QRS_NEXT_CUT()
PTP {E1 33657.188,E2 33657.188}
PTP {X 0,Y 759.907,A -85,B 0,C 180,E1 33657.188,E2 33657.188,E3 0,E4 0,E5 0,E6 0}
QRS_SPEED_INIT()
LIN {X 0,Y 759.907,Z 1240.5,A -85,B 0,C 180,E1 33657.188,E2 33657.188,E3 0,E4 0,E5 0,E6 0} C_VEL
LIN {X 0,Y 759.907,Z 488.645,A -85,B 0,C 180,E1 33657.188,E2 33657.188} C_VEL
LIN {X 0,Y 759.907,Z 480.571,A -85,B 0,C 180,E1 33657.188,E2 33657.188} C_VEL
LIN {X 0,Y 759.906,Z 478.571,A -85,B 0,C 180,E1 33657.037,E2 33657.037} C_VEL
LIN {X 0,Y 759.876,Z 478.573,A -85,B 0,C 180,E1 33654.26,E2 33654.26} C_VEL
LIN {X 0,Y 759.887,Z 478.566,A -85,B 0,C 180,E1 33651.525,E2 33651.525} C_VEL
LIN {X 0,Y 759.914,Z 478.576,A -85,B 0,C 180,E1 33648.54,E2 33648.54} C_VEL
LIN {X 0,Y 759.87,Z 478.57,A -85,B 0,C 180,E1 33645.755,E2 33645.755} C_VEL
LIN {X 0,Y 759.91,Z 478.564,A -85,B 0,C 180,E1 33643.016,E2 33643.016} C_VEL
LIN {X 0,Y 759.902,Z 478.576,A -85,B 0,C 180,E1 33640.075,E2 33640.075} C_VEL
LIN {X 0,Y 759.878,Z 478.567,A -85,B 0,C 180,E1 33637.277,E2 33637.277} C_VEL
LIN {X 0,Y 759.903,Z 478.568,A -85,B 0,C 180,E1 33634.504,E2 33634.504} C_VEL
LIN {X 0,Y 759.886,Z 478.574,A -85,B 0,C 180,E1 33631.639,E2 33631.639} C_VEL
LIN {X 0,Y 759.901,Z 478.565,A -85,B 0,C 180,E1 33628.773,E2 33628.773} C_VEL
LIN {X 0,Y 759.911,Z 478.578,A -85,B 0,C 180,E1 33625.72,E2 33625.72} C_VEL
LIN {X 0,Y 759.88,Z 478.567,A -85,B 0,C 180,E1 33622.881,E2 33622.881} C_VEL
LIN {X 0,Y 759.901,Z 478.568,A -85,B 0,C 180,E1 33620.094,E2 33620.094} C_VEL
LIN {X 0,Y 759.892,Z 478.574,A -85,B 0,C 180,E1 33617.237,E2 33617.237} C_VEL
LIN {X 0,Y 759.907,Z 478.564,A -85,B 0,C 180,E1 33614.32,E2 33614.32} C_VEL
LIN {X 0,Y 759.912,Z 478.577,A -85,B 0,C 180,E1 33611.238,E2 33611.238} C_VEL
LIN {X 0,Y 759.89,Z 478.567,A -85,B 0,C 180,E1 33608.349,E2 33608.349} C_VEL
LIN {X 0,Y 759.896,Z 478.575,A -85,B 0,C 180,E1 33605.561,E2 33605.561} C_VEL
LIN {X 0,Y 759.907,Z 478.918,A -85,B 0,C 180,E1 33605.243,E2 33605.243} C_VEL
LIN {X 0,Y 759.889,Z 515.935,A -85,B 0,C 180,E1 33603.007,E2 33603.007} C_VEL
LIN {X 0,Y 759.89,Z 560.734,A -85,B 0,C 180,E1 33600.393,E2 33600.393} C_VEL
LIN {X 0,Y 759.909,Z 611.611,A -85,B 0,C 180,E1 33597.505,E2 33597.505} C_VEL
LIN {X 0,Y 759.897,Z 651.654,A -85,B 0,C 180,E1 33595.304,E2 33595.304} C_VEL
LIN {X 0,Y 759.918,Z 925.114,A -85,B 0,C 180,E1 33592.529,E2 33592.529} C_VEL
LIN {X 0,Y 759.905,Z 958.983,A -85,B 0,C 180,E1 33592.158,E2 33592.158} C_VEL
LIN {X 0,Y 759.914,Z 979.59,A -85,B 0,C 180,E1 33591.8,E2 33591.8} C_VEL
LIN {X 0,Y 759.905,Z 1001.056,A -85,B 0,C 180,E1 33591.294,E2 33591.294} C_VEL
LIN {X 0,Y 759.917,Z 1021.303,A -85,B 0,C 180,E1 33590.686,E2 33590.686} C_VEL
LIN {X 0,Y 759.918,Z 1040.609,A -85,B 0,C 180,E1 33589.964,E2 33589.964} C_VEL
LIN {X 0,Y 759.917,Z 1060.421,A -85,B 0,C 180,E1 33589.084,E2 33589.084} C_VEL
LIN {X 0,Y 759.915,Z 1079.363,A -85,B 0,C 180,E1 33588.09,E2 33588.09} C_VEL
LIN {X 0,Y 759.915,Z 1097.201,A -85,B 0,C 180,E1 33586.983,E2 33586.983} C_VEL
LIN {X 0,Y 759.915,Z 1114.106,A -85,B 0,C 180,E1 33585.766,E2 33585.766} C_VEL
LIN {X 0,Y 759.917,Z 1129.971,A -85,B 0,C 180,E1 33584.436,E2 33584.436} C_VEL
LIN {X 0,Y 759.906,Z 1143.922,A -85,B 0,C 180,E1 33583.08,E2 33583.08} C_VEL
LIN {X 0,Y 759.906,Z 1156.086,A -85,B 0,C 180,E1 33581.691,E2 33581.691} C_VEL
LIN {X 0,Y 759.908,Z 1167.502,A -85,B 0,C 180,E1 33580.155,E2 33580.155} C_VEL
LIN {X 0,Y 759.913,Z 1177.015,A -85,B 0,C 180,E1 33578.627,E2 33578.627} C_VEL
LIN {X 0,Y 759.917,Z 1184.669,A -85,B 0,C 180,E1 33577.105,E2 33577.105} C_VEL
LIN {X 0,Y 759.909,Z 1191.249,A -85,B 0,C 180,E1 33575.436,E2 33575.436} C_VEL
LIN {X 0,Y 759.909,Z 1195.896,A -85,B 0,C 180,E1 33573.848,E2 33573.848} C_VEL
LIN {X 0,Y 759.914,Z 1198.939,A -85,B 0,C 180,E1 33572.187,E2 33572.187} C_VEL
LIN {X 0,Y 759.901,Z 1200.339,A -85,B 0,C 180,E1 33570.528,E2 33570.528} C_VEL
LIN {X 0,Y 759.911,Z 1200.186,A -85,B 0,C 180,E1 33568.945,E2 33568.945} C_VEL
LIN {X 0,Y 759.913,Z 1198.291,A -85,B 0,C 180,E1 33567.285,E2 33567.285} C_VEL
LIN {X 0,Y 759.916,Z 1194.725,A -85,B 0,C 180,E1 33565.623,E2 33565.623} C_VEL
LIN {X 0,Y 759.904,Z 1189.757,A -85,B 0,C 180,E1 33564.034,E2 33564.034} C_VEL
LIN {X 0,Y 759.899,Z 1182.966,A -85,B 0,C 180,E1 33562.439,E2 33562.439} C_VEL
LIN {X 0,Y 759.909,Z 1174.405,A -85,B 0,C 180,E1 33560.839,E2 33560.839} C_VEL
LIN {X 0,Y 759.908,Z 1164.458,A -85,B 0,C 180,E1 33559.308,E2 33559.308} C_VEL
LIN {X 0,Y 759.917,Z 1152.996,A -85,B 0,C 180,E1 33557.847,E2 33557.847} C_VEL
LIN {X 0,Y 759.915,Z 1140.229,A -85,B 0,C 180,E1 33556.455,E2 33556.455} C_VEL
LIN {X 0,Y 759.914,Z 1126.191,A -85,B 0,C 180,E1 33555.133,E2 33555.133} C_VEL
LIN {X 0,Y 759.911,Z 1110.315,A -85,B 0,C 180,E1 33553.85,E2 33553.85} C_VEL
LIN {X 0,Y 759.911,Z 1093.753,A -85,B 0,C 180,E1 33552.701,E2 33552.701} C_VEL
LIN {X 0,Y 759.917,Z 1075.204,A -85,B 0,C 180,E1 33551.592,E2 33551.592} C_VEL
LIN {X 0,Y 759.917,Z 1056.495,A -85,B 0,C 180,E1 33550.635,E2 33550.635} C_VEL
LIN {X 0,Y 759.92,Z 1036.873,A -85,B 0,C 180,E1 33549.795,E2 33549.795} C_VEL
LIN {X 0,Y 759.916,Z 1016.314,A -85,B 0,C 180,E1 33549.066,E2 33549.066} C_VEL
LIN {X 0,Y 759.911,Z 995.942,A -85,B 0,C 180,E1 33548.478,E2 33548.478} C_VEL
LIN {X 0,Y 759.909,Z 974.842,A -85,B 0,C 180,E1 33548.017,E2 33548.017} C_VEL
LIN {X 0,Y 759.907,Z 952.592,A -85,B 0,C 180,E1 33547.671,E2 33547.671} C_VEL
LIN {X 0,Y 759.898,Z 670.991,A -85,B 0,C 180,E1 33544.808,E2 33544.808} C_VEL
LIN {X 0,Y 759.898,Z 651.373,A -85,B 0,C 180,E1 33544.6,E2 33544.6} C_VEL
LIN {X 0,Y 759.905,Z 601.06,A -85,B 0,C 180,E1 33541.812,E2 33541.812} C_VEL
LIN {X 0,Y 759.918,Z 552.419,A -85,B 0,C 180,E1 33539.039,E2 33539.039} C_VEL
LIN {X 0,Y 759.919,Z 505.108,A -85,B 0,C 180,E1 33536.261,E2 33536.261} C_VEL
LIN {X 0,Y 759.908,Z 478.918,A -85,B 0,C 180,E1 33534.667,E2 33534.667} C_VEL
LIN {X 0,Y 759.908,Z 478.57,A -85,B 0,C 180,E1 33534.149,E2 33534.149} C_VEL
LIN {X 0,Y 759.874,Z 478.571,A -85,B 0,C 180,E1 33531.317,E2 33531.317} C_VEL
LIN {X 0,Y 759.914,Z 478.576,A -85,B 0,C 180,E1 33528.561,E2 33528.561} C_VEL
LIN {X 0,Y 759.894,Z 478.566,A -85,B 0,C 180,E1 33525.573,E2 33525.573} C_VEL
LIN {X 0,Y 759.884,Z 478.573,A -85,B 0,C 180,E1 33522.759,E2 33522.759} C_VEL
LIN {X 0,Y 759.904,Z 478.569,A -85,B 0,C 180,E1 33519.907,E2 33519.907} C_VEL
LIN {X 0,Y 759.877,Z 478.567,A -85,B 0,C 180,E1 33517.119,E2 33517.119} C_VEL
LIN {X 0,Y 759.895,Z 478.576,A -85,B 0,C 180,E1 33514.367,E2 33514.367} C_VEL
LIN {X 0,Y 759.91,Z 478.564,A -85,B 0,C 180,E1 33511.315,E2 33511.315} C_VEL
LIN {X 0,Y 759.868,Z 478.571,A -85,B 0,C 180,E1 33508.619,E2 33508.619} C_VEL
LIN {X 0,Y 759.912,Z 478.576,A -85,B 0,C 180,E1 33505.845,E2 33505.845} C_VEL
LIN {X 0,Y 759.891,Z 478.565,A -85,B 0,C 180,E1 33502.92,E2 33502.92} C_VEL
LIN {X 0,Y 759.874,Z 478.573,A -85,B 0,C 180,E1 33500.167,E2 33500.167} C_VEL
LIN {X 0,Y 759.906,Z 478.572,A -85,B 0,C 180,E1 33497.379,E2 33497.379} C_VEL
LIN {X 0,Y 759.878,Z 478.567,A -85,B 0,C 180,E1 33494.556,E2 33494.556} C_VEL
LIN {X 0,Y 759.877,Z 478.574,A -85,B 0,C 180,E1 33491.846,E2 33491.846} C_VEL
LIN {X 0,Y 759.907,Z 478.569,A -85,B 0,C 180,E1 33489.009,E2 33489.009} C_VEL
LIN {X 0,Y 759.868,Z 478.568,A -85,B 0,C 180,E1 33486.194,E2 33486.194} C_VEL
LIN {X 0,Y 759.887,Z 478.575,A -85,B 0,C 180,E1 33483.47,E2 33483.47} C_VEL
LIN {X 0,Y 759.91,Z 478.565,A -85,B 0,C 180,E1 33480.452,E2 33480.452} C_VEL
LIN {X 0,Y 759.861,Z 478.571,A -85,B 0,C 180,E1 33477.738,E2 33477.738} C_VEL
LIN {X 0,Y 759.909,Z 478.577,A -85,B 0,C 180,E1 33475.018,E2 33475.018} C_VEL
LIN {X 0,Y 759.888,Z 478.566,A -85,B 0,C 180,E1 33472.058,E2 33472.058} C_VEL
LIN {X 0,Y 759.861,Z 478.572,A -85,B 0,C 180,E1 33469.384,E2 33469.384} C_VEL
LIN {X 0,Y 759.918,Z 478.577,A -85,B 0,C 180,E1 33466.687,E2 33466.687} C_VEL
LIN {X 0,Y 759.876,Z 478.567,A -85,B 0,C 180,E1 33463.723,E2 33463.723} C_VEL
LIN {X 0,Y 759.86,Z 478.573,A -85,B 0,C 180,E1 33461.101,E2 33461.101} C_VEL
LIN {X 0,Y 759.915,Z 478.576,A -85,B 0,C 180,E1 33458.382,E2 33458.382} C_VEL
LIN {X 0,Y 759.877,Z 478.567,A -85,B 0,C 180,E1 33455.512,E2 33455.512} C_VEL
LIN {X 0,Y 759.856,Z 478.572,A -85,B 0,C 180,E1 33452.916,E2 33452.916} C_VEL
LIN {X 0,Y 759.904,Z 478.578,A -85,B 0,C 180,E1 33450.26,E2 33450.26} C_VEL
LIN {X 0,Y 759.883,Z 478.566,A -85,B 0,C 180,E1 33447.35,E2 33447.35} C_VEL
LIN {X 0,Y 759.853,Z 478.572,A -85,B 0,C 180,E1 33444.712,E2 33444.712} C_VEL
LIN {X 0,Y 759.914,Z 478.577,A -85,B 0,C 180,E1 33441.99,E2 33441.99} C_VEL
LIN {X 0,Y 759.874,Z 478.568,A -85,B 0,C 180,E1 33439.05,E2 33439.05} C_VEL
LIN {X 0,Y 759.851,Z 478.572,A -85,B 0,C 180,E1 33436.472,E2 33436.472} C_VEL
LIN {X 0,Y 759.912,Z 478.577,A -85,B 0,C 180,E1 33433.749,E2 33433.749} C_VEL
LIN {X 0,Y 759.875,Z 478.569,A -85,B 0,C 180,E1 33430.832,E2 33430.832} C_VEL
LIN {X 0,Y 759.849,Z 478.573,A -85,B 0,C 180,E1 33428.224,E2 33428.224} C_VEL
LIN {X 0,Y 759.889,Z 478.702,A -85,B 0,C 180,E1 33425.639,E2 33425.639} C_VEL
LIN {X 0,Y 759.917,Z 480.91,A -85,B 0,C 180,E1 33425.464,E2 33425.464} C_VEL
LIN {X 0,Y 759.915,Z 527.036,A -85,B 0,C 180,E1 33422.87,E2 33422.87} C_VEL
LIN {X 0,Y 759.912,Z 529.446,A -85,B 0,C 180,E1 33422.801,E2 33422.801} C_VEL
LIN {X 0,Y 759.891,Z 789.76,A -85,B 0,C 180,E1 33419.978,E2 33419.978} C_VEL
LIN {X 0,Y 759.917,Z 918.081,A -85,B 0,C 180,E1 33418.594,E2 33418.594} C_VEL
LIN {X 0,Y 759.894,Z 942.353,A -85,B 0,C 180,E1 33418.209,E2 33418.209} C_VEL
LIN {X 0,Y 759.901,Z 963.718,A -85,B 0,C 180,E1 33417.741,E2 33417.741} C_VEL
LIN {X 0,Y 759.907,Z 983.081,A -85,B 0,C 180,E1 33417.221,E2 33417.221} C_VEL
LIN {X 0,Y 759.919,Z 1005.766,A -85,B 0,C 180,E1 33416.49,E2 33416.49} C_VEL
LIN {X 0,Y 759.916,Z 1027.274,A -85,B 0,C 180,E1 33415.65,E2 33415.65} C_VEL
LIN {X 0,Y 759.918,Z 1046.636,A -85,B 0,C 180,E1 33414.784,E2 33414.784} C_VEL
LIN {X 0,Y 759.909,Z 1068.349,A -85,B 0,C 180,E1 33413.66,E2 33413.66} C_VEL
LIN {X 0,Y 759.913,Z 1086.397,A -85,B 0,C 180,E1 33412.594,E2 33412.594} C_VEL
LIN {X 0,Y 759.907,Z 1107.535,A -85,B 0,C 180,E1 33411.172,E2 33411.172} C_VEL
LIN {X 0,Y 759.916,Z 1124.895,A -85,B 0,C 180,E1 33409.844,E2 33409.844} C_VEL
LIN {X 0,Y 759.916,Z 1141.398,A -85,B 0,C 180,E1 33408.408,E2 33408.408} C_VEL
LIN {X 0,Y 759.898,Z 1155.953,A -85,B 0,C 180,E1 33406.984,E2 33406.984} C_VEL
LIN {X 0,Y 759.899,Z 1170.876,A -85,B 0,C 180,E1 33405.312,E2 33405.312} C_VEL
LIN {X 0,Y 759.9,Z 1182.583,A -85,B 0,C 180,E1 33403.813,E2 33403.813} C_VEL
LIN {X 0,Y 759.894,Z 1194.788,A -85,B 0,C 180,E1 33401.999,E2 33401.999} C_VEL
LIN {X 0,Y 759.907,Z 1203.557,A -85,B 0,C 180,E1 33400.462,E2 33400.462} C_VEL
LIN {X 0,Y 759.894,Z 1212.075,A -85,B 0,C 180,E1 33398.703,E2 33398.703} C_VEL
LIN {X 0,Y 759.918,Z 1218.727,A -85,B 0,C 180,E1 33396.953,E2 33396.953} C_VEL
LIN {X 0,Y 759.883,Z 1223.511,A -85,B 0,C 180,E1 33395.36,E2 33395.36} C_VEL
LIN {X 0,Y 759.919,Z 1227.559,A -85,B 0,C 180,E1 33393.47,E2 33393.47} C_VEL
LIN {X 0,Y 759.9,Z 1229.63,A -85,B 0,C 180,E1 33391.81,E2 33391.81} C_VEL
LIN {X 0,Y 759.92,Z 1230.5,A -85,B 0,C 180,E1 33390,E2 33390} C_VEL
LIN {X 0,Y 759.9,Z 1229.63,A -85,B 0,C 180,E1 33388.19,E2 33388.19} C_VEL
LIN {X 0,Y 759.919,Z 1227.559,A -85,B 0,C 180,E1 33386.53,E2 33386.53} C_VEL
LIN {X 0,Y 759.883,Z 1223.511,A -85,B 0,C 180,E1 33384.639,E2 33384.639} C_VEL
LIN {X 0,Y 759.918,Z 1218.726,A -85,B 0,C 180,E1 33383.047,E2 33383.047} C_VEL
LIN {X 0,Y 759.893,Z 1211.731,A -85,B 0,C 180,E1 33381.221,E2 33381.221} C_VEL
LIN {X 0,Y 759.907,Z 1203.557,A -85,B 0,C 180,E1 33379.538,E2 33379.538} C_VEL
LIN {X 0,Y 759.894,Z 1194.788,A -85,B 0,C 180,E1 33378.001,E2 33378.001} C_VEL
LIN {X 0,Y 759.9,Z 1182.583,A -85,B 0,C 180,E1 33376.187,E2 33376.187} C_VEL
LIN {X 0,Y 759.899,Z 1170.876,A -85,B 0,C 180,E1 33374.688,E2 33374.688} C_VEL
LIN {X 0,Y 759.898,Z 1155.953,A -85,B 0,C 180,E1 33373.016,E2 33373.016} C_VEL
LIN {X 0,Y 759.916,Z 1141.398,A -85,B 0,C 180,E1 33371.592,E2 33371.592} C_VEL
LIN {X 0,Y 759.911,Z 1123.375,A -85,B 0,C 180,E1 33370.036,E2 33370.036} C_VEL
LIN {X 0,Y 759.908,Z 1106.43,A -85,B 0,C 180,E1 33368.747,E2 33368.747} C_VEL
LIN {X 0,Y 759.914,Z 1086.396,A -85,B 0,C 180,E1 33367.406,E2 33367.406} C_VEL
LIN {X 0,Y 759.909,Z 1067.993,A -85,B 0,C 180,E1 33366.32,E2 33366.32} C_VEL
LIN {X 0,Y 759.919,Z 1045.919,A -85,B 0,C 180,E1 33365.183,E2 33365.183} C_VEL
LIN {X 0,Y 759.916,Z 1026.866,A -85,B 0,C 180,E1 33364.332,E2 33364.332} C_VEL
LIN {X 0,Y 759.918,Z 1004.811,A -85,B 0,C 180,E1 33363.475,E2 33363.475} C_VEL
LIN {X 0,Y 759.907,Z 982.044,A -85,B 0,C 180,E1 33362.749,E2 33362.749} C_VEL
LIN {X 0,Y 759.898,Z 962.099,A -85,B 0,C 180,E1 33362.219,E2 33362.219} C_VEL
LIN {X 0,Y 759.898,Z 937.439,A -85,B 0,C 180,E1 33361.702,E2 33361.702} C_VEL
LIN {X 0,Y 759.916,Z 916.368,A -85,B 0,C 180,E1 33361.384,E2 33361.384} C_VEL
LIN {X 0,Y 759.867,Z 652.343,A -85,B 0,C 180,E1 33358.541,E2 33358.541} C_VEL
LIN {X 0,Y 759.912,Z 527.915,A -85,B 0,C 180,E1 33357.174,E2 33357.174} C_VEL
LIN {X 0,Y 759.916,Z 481.69,A -85,B 0,C 180,E1 33354.58,E2 33354.58} C_VEL
LIN {X 0,Y 759.891,Z 478.77,A -85,B 0,C 180,E1 33354.377,E2 33354.377} C_VEL
LIN {X 0,Y 759.852,Z 478.574,A -85,B 0,C 180,E1 33351.893,E2 33351.893} C_VEL
LIN {X 0,Y 759.858,Z 478.57,A -85,B 0,C 180,E1 33349.357,E2 33349.357} C_VEL
LIN {X 0,Y 759.913,Z 478.57,A -85,B 0,C 180,E1 33346.579,E2 33346.579} C_VEL
LIN {X 0,Y 759.861,Z 478.573,A -85,B 0,C 180,E1 33343.747,E2 33343.747} C_VEL
LIN {X 0,Y 759.859,Z 478.57,A -85,B 0,C 180,E1 33341.144,E2 33341.144} C_VEL
LIN {X 0,Y 759.911,Z 478.569,A -85,B 0,C 180,E1 33338.354,E2 33338.354} C_VEL
LIN {X 0,Y 759.868,Z 478.574,A -85,B 0,C 180,E1 33335.564,E2 33335.564} C_VEL
LIN {X 0,Y 759.861,Z 478.568,A -85,B 0,C 180,E1 33332.92,E2 33332.92} C_VEL
LIN {X 0,Y 759.912,Z 478.569,A -85,B 0,C 180,E1 33330.175,E2 33330.175} C_VEL
LIN {X 0,Y 759.873,Z 478.574,A -85,B 0,C 180,E1 33327.338,E2 33327.338} C_VEL
LIN {X 0,Y 759.861,Z 478.569,A -85,B 0,C 180,E1 33324.737,E2 33324.737} C_VEL
LIN {X 0,Y 759.915,Z 478.567,A -85,B 0,C 180,E1 33322.024,E2 33322.024} C_VEL
LIN {X 0,Y 759.878,Z 478.575,A -85,B 0,C 180,E1 33319.126,E2 33319.126} C_VEL
LIN {X 0,Y 759.866,Z 478.569,A -85,B 0,C 180,E1 33316.434,E2 33316.434} C_VEL
LIN {X 0,Y 759.91,Z 478.568,A -85,B 0,C 180,E1 33313.7,E2 33313.7} C_VEL
LIN {X 0,Y 759.878,Z 478.574,A -85,B 0,C 180,E1 33310.846,E2 33310.846} C_VEL
LIN {X 0,Y 759.87,Z 478.568,A -85,B 0,C 180,E1 33308.17,E2 33308.17} C_VEL
LIN {X 0,Y 759.907,Z 478.57,A -85,B 0,C 180,E1 33305.361,E2 33305.361} C_VEL
LIN {X 0,Y 759.877,Z 478.574,A -85,B 0,C 180,E1 33302.564,E2 33302.564} C_VEL
LIN {X 0,Y 759.877,Z 478.567,A -85,B 0,C 180,E1 33299.849,E2 33299.849} C_VEL
LIN {X 0,Y 759.906,Z 478.571,A -85,B 0,C 180,E1 33297.037,E2 33297.037} C_VEL
LIN {X 0,Y 758.93,Z 478.703,A -85,B 0,C 180,E1 33296.456,E2 33296.456} C_VEL
LIN {X 0,Y 752.51,Z 479.501,A -85,B 0,C 180,E1 33294.83,E2 33294.83} C_VEL
LIN {X 0,Y 751.949,Z 479.563,A -85,B 0,C 180,E1 33294.407,E2 33294.407} C_VEL
LIN {X 0,Y 751.942,Z 479.556,A -85,B 0,C 180,E1 33291.589,E2 33291.589} C_VEL
LIN {X 0,Y 751.967,Z 479.56,A -85,B 0,C 180,E1 33288.728,E2 33288.728} C_VEL
LIN {X 0,Y 751.934,Z 479.56,A -85,B 0,C 180,E1 33285.916,E2 33285.916} C_VEL
LIN {X 0,Y 751.972,Z 479.553,A -85,B 0,C 180,E1 33283.07,E2 33283.07} C_VEL
LIN {X 0,Y 751.957,Z 479.564,A -85,B 0,C 180,E1 33280.017,E2 33280.017} C_VEL
LIN {X 0,Y 751.942,Z 479.555,A -85,B 0,C 180,E1 33277.235,E2 33277.235} C_VEL
LIN {X 0,Y 751.964,Z 479.559,A -85,B 0,C 180,E1 33274.396,E2 33274.396} C_VEL
LIN {X 0,Y 751.943,Z 479.562,A -85,B 0,C 180,E1 33271.572,E2 33271.572} C_VEL
LIN {X 0,Y 751.964,Z 479.553,A -85,B 0,C 180,E1 33268.756,E2 33268.756} C_VEL
LIN {X 0,Y 751.968,Z 479.566,A -85,B 0,C 180,E1 33265.661,E2 33265.661} C_VEL
LIN {X 0,Y 751.948,Z 479.553,A -85,B 0,C 180,E1 33262.769,E2 33262.769} C_VEL
LIN {X 0,Y 751.961,Z 479.559,A -85,B 0,C 180,E1 33259.94,E2 33259.94} C_VEL
LIN {X 0,Y 751.95,Z 479.561,A -85,B 0,C 180,E1 33257.196,E2 33257.196} C_VEL
LIN {X 0,Y 751.974,Z 479.553,A -85,B 0,C 180,E1 33254.272,E2 33254.272} C_VEL
LIN {X 0,Y 751.967,Z 479.565,A -85,B 0,C 180,E1 33251.183,E2 33251.183} C_VEL
LIN {X 0,Y 751.964,Z 479.556,A -85,B 0,C 180,E1 33248.191,E2 33248.191} C_VEL
LIN {X 0,Y 751.982,Z 479.737,A -85,B 0,C 180,E1 33245.641,E2 33245.641} C_VEL
LIN {X 0,Y 752.908,Z 483.22,A -85,B 0,C 180,E1 33245.339,E2 33245.339} C_VEL
LIN {X 0,Y 752.739,Z 526.575,A -85,B 0,C 180,E1 33242.725,E2 33242.725} C_VEL
LIN {X 0,Y 752.644,Z 573.653,A -85,B 0,C 180,E1 33239.967,E2 33239.967} C_VEL
LIN {X 0,Y 752.503,Z 622.252,A -85,B 0,C 180,E1 33237.199,E2 33237.199} C_VEL
LIN {X 0,Y 752.525,Z 651.817,A -85,B 0,C 180,E1 33235.568,E2 33235.568} C_VEL
LIN {X 0,Y 752.566,Z 857.23,A -85,B 0,C 180,E1 33233.452,E2 33233.452} C_VEL
LIN {X 0,Y 752.494,Z 956.636,A -85,B 0,C 180,E1 33232.422,E2 33232.422} C_VEL
LIN {X 0,Y 752.461,Z 977.93,A -85,B 0,C 180,E1 33232.061,E2 33232.061} C_VEL
LIN {X 0,Y 752.403,Z 999.609,A -85,B 0,C 180,E1 33231.558,E2 33231.558} C_VEL
LIN {X 0,Y 752.372,Z 1019.992,A -85,B 0,C 180,E1 33230.946,E2 33230.946} C_VEL
LIN {X 0,Y 752.309,Z 1039.631,A -85,B 0,C 180,E1 33230.216,E2 33230.216} C_VEL
LIN {X 0,Y 752.24,Z 1059.632,A -85,B 0,C 180,E1 33229.327,E2 33229.327} C_VEL
LIN {X 0,Y 752.187,Z 1078.654,A -85,B 0,C 180,E1 33228.323,E2 33228.323} C_VEL
LIN {X 0,Y 752.125,Z 1096.369,A -85,B 0,C 180,E1 33227.22,E2 33227.22} C_VEL
LIN {X 0,Y 752.074,Z 1113.607,A -85,B 0,C 180,E1 33225.974,E2 33225.974} C_VEL
LIN {X 0,Y 752.028,Z 1128.683,A -85,B 0,C 180,E1 33224.711,E2 33224.711} C_VEL
LIN {X 0,Y 751.996,Z 1142.434,A -85,B 0,C 180,E1 33223.377,E2 33223.377} C_VEL
LIN {X 0,Y 751.967,Z 1154.812,A -85,B 0,C 180,E1 33221.972,E2 33221.972} C_VEL
LIN {X 0,Y 751.944,Z 1166.471,A -85,B 0,C 180,E1 33220.419,E2 33220.419} C_VEL
LIN {X 0,Y 751.93,Z 1176.168,A -85,B 0,C 180,E1 33218.873,E2 33218.873} C_VEL
LIN {X 0,Y 751.914,Z 1183.964,A -85,B 0,C 180,E1 33217.334,E2 33217.334} C_VEL
LIN {X 0,Y 751.9,Z 1190.492,A -85,B 0,C 180,E1 33215.724,E2 33215.724} C_VEL
LIN {X 0,Y 751.918,Z 1195.302,A -85,B 0,C 180,E1 33214.118,E2 33214.118} C_VEL
LIN {X 0,Y 751.911,Z 1198.606,A -85,B 0,C 180,E1 33212.439,E2 33212.439} C_VEL
LIN {X 0,Y 751.913,Z 1200.272,A -85,B 0,C 180,E1 33210.762,E2 33210.762} C_VEL
LIN {X 0,Y 751.913,Z 1200.254,A -85,B 0,C 180,E1 33209.086,E2 33209.086} C_VEL
LIN {X 0,Y 751.909,Z 1198.626,A -85,B 0,C 180,E1 33207.485,E2 33207.485} C_VEL
LIN {X 0,Y 751.918,Z 1195.338,A -85,B 0,C 180,E1 33205.806,E2 33205.806} C_VEL
LIN {X 0,Y 751.904,Z 1190.536,A -85,B 0,C 180,E1 33204.2,E2 33204.2} C_VEL
LIN {X 0,Y 751.911,Z 1184.025,A -85,B 0,C 180,E1 33202.589,E2 33202.589} C_VEL
LIN {X 0,Y 751.931,Z 1176.245,A -85,B 0,C 180,E1 33201.05,E2 33201.05} C_VEL
LIN {X 0,Y 751.945,Z 1166.555,A -85,B 0,C 180,E1 33199.504,E2 33199.504} C_VEL
LIN {X 0,Y 751.964,Z 1154.912,A -85,B 0,C 180,E1 33197.951,E2 33197.951} C_VEL
LIN {X 0,Y 751.997,Z 1142.549,A -85,B 0,C 180,E1 33196.545,E2 33196.545} C_VEL
LIN {X 0,Y 752.028,Z 1128.199,A -85,B 0,C 180,E1 33195.154,E2 33195.154} C_VEL
LIN {X 0,Y 752.071,Z 1112.734,A -85,B 0,C 180,E1 33193.868,E2 33193.868} C_VEL
LIN {X 0,Y 752.124,Z 1095.859,A -85,B 0,C 180,E1 33192.656,E2 33192.656} C_VEL
LIN {X 0,Y 752.189,Z 1078.106,A -85,B 0,C 180,E1 33191.557,E2 33191.557} C_VEL
LIN {X 0,Y 752.24,Z 1059.818,A -85,B 0,C 180,E1 33190.592,E2 33190.592} C_VEL
LIN {X 0,Y 752.309,Z 1039.849,A -85,B 0,C 180,E1 33189.703,E2 33189.703} C_VEL
LIN {X 0,Y 752.37,Z 1020.259,A -85,B 0,C 180,E1 33188.973,E2 33188.973} C_VEL
LIN {X 0,Y 752.403,Z 999.9,A -85,B 0,C 180,E1 33188.361,E2 33188.361} C_VEL
LIN {X 0,Y 752.461,Z 977.95,A -85,B 0,C 180,E1 33187.85,E2 33187.85} C_VEL
LIN {X 0,Y 752.494,Z 956.737,A -85,B 0,C 180,E1 33187.489,E2 33187.489} C_VEL
LIN {X 0,Y 752.563,Z 860.44,A -85,B 0,C 180,E1 33186.491,E2 33186.491} C_VEL
LIN {X 0,Y 752.538,Z 651.902,A -85,B 0,C 180,E1 33184.344,E2 33184.344} C_VEL
LIN {X 0,Y 752.461,Z 636.009,A -85,B 0,C 180,E1 33183.483,E2 33183.483} C_VEL
LIN {X 0,Y 752.565,Z 589.65,A -85,B 0,C 180,E1 33180.861,E2 33180.861} C_VEL
LIN {X 0,Y 752.723,Z 541.008,A -85,B 0,C 180,E1 33178.039,E2 33178.039} C_VEL
LIN {X 0,Y 752.872,Z 494.644,A -85,B 0,C 180,E1 33175.268,E2 33175.268} C_VEL
LIN {X 0,Y 752.808,Z 482.281,A -85,B 0,C 180,E1 33174.508,E2 33174.508} C_VEL
LIN {X 0,Y 751.986,Z 479.719,A -85,B 0,C 180,E1 33174.265,E2 33174.265} C_VEL
LIN {X 0,Y 751.937,Z 479.56,A -85,B 0,C 180,E1 33171.435,E2 33171.435} C_VEL
LIN {X 0,Y 751.973,Z 479.567,A -85,B 0,C 180,E1 33168.637,E2 33168.637} C_VEL
LIN {X 0,Y 751.96,Z 479.554,A -85,B 0,C 180,E1 33165.621,E2 33165.621} C_VEL
LIN {X 0,Y 751.944,Z 479.561,A -85,B 0,C 180,E1 33162.778,E2 33162.778} C_VEL
LIN {X 0,Y 751.965,Z 479.559,A -85,B 0,C 180,E1 33159.96,E2 33159.96} C_VEL
LIN {X 0,Y 751.939,Z 479.554,A -85,B 0,C 180,E1 33157.136,E2 33157.136} C_VEL
LIN {X 0,Y 751.961,Z 479.565,A -85,B 0,C 180,E1 33154.319,E2 33154.319} C_VEL
LIN {X 0,Y 751.963,Z 479.554,A -85,B 0,C 180,E1 33151.238,E2 33151.238} C_VEL
LIN {X 0,Y 751.934,Z 479.562,A -85,B 0,C 180,E1 33148.428,E2 33148.428} C_VEL
LIN {X 0,Y 751.966,Z 479.56,A -85,B 0,C 180,E1 33145.604,E2 33145.604} C_VEL
LIN {X 0,Y 751.939,Z 479.556,A -85,B 0,C 180,E1 33142.765,E2 33142.765} C_VEL
LIN {X 0,Y 751.949,Z 479.564,A -85,B 0,C 180,E1 33139.983,E2 33139.983} C_VEL
LIN {X 0,Y 751.973,Z 479.554,A -85,B 0,C 180,E1 33137.01,E2 33137.01} C_VEL
LIN {X 0,Y 751.927,Z 479.559,A -85,B 0,C 180,E1 33134.218,E2 33134.218} C_VEL
LIN {X 0,Y 751.977,Z 479.564,A -85,B 0,C 180,E1 33131.427,E2 33131.427} C_VEL
LIN {X 0,Y 751.948,Z 479.556,A -85,B 0,C 180,E1 33128.488,E2 33128.488} C_VEL
LIN {X 0,Y 751.929,Z 479.561,A -85,B 0,C 180,E1 33125.8,E2 33125.8} C_VEL
LIN {X 0,Y 751.972,Z 479.562,A -85,B 0,C 180,E1 33123.049,E2 33123.049} C_VEL
LIN {X 0,Y 751.937,Z 479.556,A -85,B 0,C 180,E1 33120.152,E2 33120.152} C_VEL
LIN {X 0,Y 751.93,Z 479.562,A -85,B 0,C 180,E1 33117.485,E2 33117.485} C_VEL
LIN {X 0,Y 751.97,Z 479.56,A -85,B 0,C 180,E1 33114.659,E2 33114.659} C_VEL
LIN {X 0,Y 751.934,Z 479.556,A -85,B 0,C 180,E1 33111.897,E2 33111.897} C_VEL
LIN {X 0,Y 751.932,Z 479.563,A -85,B 0,C 180,E1 33109.193,E2 33109.193} C_VEL
LIN {X 0,Y 751.972,Z 479.558,A -85,B 0,C 180,E1 33106.309,E2 33106.309} C_VEL
LIN {X 0,Y 751.924,Z 479.558,A -85,B 0,C 180,E1 33103.546,E2 33103.546} C_VEL
LIN {X 0,Y 751.933,Z 479.563,A -85,B 0,C 180,E1 33100.906,E2 33100.906} C_VEL
LIN {X 0,Y 751.978,Z 479.555,A -85,B 0,C 180,E1 33097.934,E2 33097.934} C_VEL
LIN {X 0,Y 751.919,Z 479.558,A -85,B 0,C 180,E1 33095.236,E2 33095.236} C_VEL
LIN {X 0,Y 751.936,Z 479.564,A -85,B 0,C 180,E1 33092.607,E2 33092.607} C_VEL
LIN {X 0,Y 751.974,Z 479.555,A -85,B 0,C 180,E1 33089.648,E2 33089.648} C_VEL
LIN {X 0,Y 751.915,Z 479.557,A -85,B 0,C 180,E1 33086.902,E2 33086.902} C_VEL
LIN {X 0,Y 751.954,Z 479.565,A -85,B 0,C 180,E1 33084.191,E2 33084.191} C_VEL
LIN {X 0,Y 751.944,Z 479.553,A -85,B 0,C 180,E1 33081.187,E2 33081.187} C_VEL
LIN {X 0,Y 751.912,Z 479.561,A -85,B 0,C 180,E1 33078.589,E2 33078.589} C_VEL
LIN {X 0,Y 751.969,Z 479.563,A -85,B 0,C 180,E1 33075.832,E2 33075.832} C_VEL
LIN {X 0,Y 751.936,Z 479.556,A -85,B 0,C 180,E1 33072.887,E2 33072.887} C_VEL
LIN {X 0,Y 751.911,Z 479.562,A -85,B 0,C 180,E1 33070.36,E2 33070.36} C_VEL
LIN {X 0,Y 751.95,Z 479.568,A -85,B 0,C 180,E1 33067.703,E2 33067.703} C_VEL
LIN {X 0,Y 751.951,Z 479.807,A -85,B 0,C 180,E1 33065.989,E2 33065.989} C_VEL
LIN {X 0,Y 752.966,Z 483.28,A -85,B 0,C 180,E1 33065.705,E2 33065.705} C_VEL
LIN {X 0,Y 752.93,Z 528.408,A -85,B 0,C 180,E1 33063.159,E2 33063.159} C_VEL
LIN {X 0,Y 753.173,Z 534.727,A -85,B 0,C 180,E1 33063.073,E2 33063.073} C_VEL
LIN {X 0,Y 752.954,Z 792.05,A -85,B 0,C 180,E1 33060.258,E2 33060.258} C_VEL
LIN {X 0,Y 752.881,Z 918.509,A -85,B 0,C 180,E1 33058.881,E2 33058.881} C_VEL
LIN {X 0,Y 752.797,Z 943.511,A -85,B 0,C 180,E1 33058.475,E2 33058.475} C_VEL
LIN {X 0,Y 752.753,Z 964.643,A -85,B 0,C 180,E1 33058.005,E2 33058.005} C_VEL
LIN {X 0,Y 752.701,Z 985.717,A -85,B 0,C 180,E1 33057.426,E2 33057.426} C_VEL
LIN {X 0,Y 752.612,Z 1010.071,A -85,B 0,C 180,E1 33056.604,E2 33056.604} C_VEL
LIN {X 0,Y 752.542,Z 1029.266,A -85,B 0,C 180,E1 33055.836,E2 33055.836} C_VEL
LIN {X 0,Y 752.446,Z 1051.242,A -85,B 0,C 180,E1 33054.823,E2 33054.823} C_VEL
LIN {X 0,Y 752.361,Z 1071.26,A -85,B 0,C 180,E1 33053.745,E2 33053.745} C_VEL
LIN {X 0,Y 752.275,Z 1091.613,A -85,B 0,C 180,E1 33052.506,E2 33052.506} C_VEL
LIN {X 0,Y 752.196,Z 1110.297,A -85,B 0,C 180,E1 33051.196,E2 33051.196} C_VEL
LIN {X 0,Y 752.117,Z 1128.753,A -85,B 0,C 180,E1 33049.735,E2 33049.735} C_VEL
LIN {X 0,Y 752.079,Z 1144.801,A -85,B 0,C 180,E1 33048.285,E2 33048.285} C_VEL
LIN {X 0,Y 752.026,Z 1161.096,A -85,B 0,C 180,E1 33046.61,E2 33046.61} C_VEL
LIN {X 0,Y 751.972,Z 1173.894,A -85,B 0,C 180,E1 33045.106,E2 33045.106} C_VEL
LIN {X 0,Y 751.94,Z 1187.234,A -85,B 0,C 180,E1 33043.299,E2 33043.299} C_VEL
LIN {X 0,Y 751.925,Z 1196.64,A -85,B 0,C 180,E1 33041.816,E2 33041.816} C_VEL
LIN {X 0,Y 751.907,Z 1206.401,A -85,B 0,C 180,E1 33040.032,E2 33040.032} C_VEL
LIN {X 0,Y 751.926,Z 1214.207,A -85,B 0,C 180,E1 33038.257,E2 33038.257} C_VEL
LIN {X 0,Y 751.908,Z 1220.135,A -85,B 0,C 180,E1 33036.602,E2 33036.602} C_VEL
LIN {X 0,Y 751.915,Z 1225.336,A -85,B 0,C 180,E1 33034.653,E2 33034.653} C_VEL
LIN {X 0,Y 751.884,Z 1228.234,A -85,B 0,C 180,E1 33033.049,E2 33033.049} C_VEL
LIN {X 0,Y 751.913,Z 1230.15,A -85,B 0,C 180,E1 33031.219,E2 33031.219} C_VEL
LIN {X 0,Y 751.881,Z 1230.351,A -85,B 0,C 180,E1 33029.467,E2 33029.467} C_VEL
LIN {X 0,Y 751.919,Z 1229.296,A -85,B 0,C 180,E1 33027.79,E2 33027.79} C_VEL
LIN {X 0,Y 751.917,Z 1226.288,A -85,B 0,C 180,E1 33025.806,E2 33025.806} C_VEL
LIN {X 0,Y 751.918,Z 1222.482,A -85,B 0,C 180,E1 33024.2,E2 33024.2} C_VEL
LIN {X 0,Y 751.889,Z 1216.638,A -85,B 0,C 180,E1 33022.358,E2 33022.358} C_VEL
LIN {X 0,Y 751.919,Z 1209.523,A -85,B 0,C 180,E1 33020.647,E2 33020.647} C_VEL
LIN {X 0,Y 751.905,Z 1201.518,A -85,B 0,C 180,E1 33019.038,E2 33019.038} C_VEL
LIN {X 0,Y 751.937,Z 1190.353,A -85,B 0,C 180,E1 33017.17,E2 33017.17} C_VEL
LIN {X 0,Y 751.963,Z 1179.954,A -85,B 0,C 180,E1 33015.681,E2 33015.681} C_VEL
LIN {X 0,Y 751.998,Z 1166.68,A -85,B 0,C 180,E1 33014.016,E2 33014.016} C_VEL
LIN {X 0,Y 752.052,Z 1152.848,A -85,B 0,C 180,E1 33012.514,E2 33012.514} C_VEL
LIN {X 0,Y 752.113,Z 1136.635,A -85,B 0,C 180,E1 33010.951,E2 33010.951} C_VEL
LIN {X 0,Y 752.156,Z 1119.829,A -85,B 0,C 180,E1 33009.536,E2 33009.536} C_VEL
LIN {X 0,Y 752.241,Z 1100.444,A -85,B 0,C 180,E1 33008.094,E2 33008.094} C_VEL
LIN {X 0,Y 752.311,Z 1082.43,A -85,B 0,C 180,E1 33006.917,E2 33006.917} C_VEL
LIN {X 0,Y 752.415,Z 1060.765,A -85,B 0,C 180,E1 33005.673,E2 33005.673} C_VEL
LIN {X 0,Y 752.487,Z 1041.473,A -85,B 0,C 180,E1 33004.711,E2 33004.711} C_VEL
LIN {X 0,Y 752.594,Z 1019.167,A -85,B 0,C 180,E1 33003.741,E2 33003.741} C_VEL
LIN {X 0,Y 752.662,Z 998.264,A -85,B 0,C 180,E1 33002.979,E2 33002.979} C_VEL
LIN {X 0,Y 752.716,Z 979.03,A -85,B 0,C 180,E1 33002.379,E2 33002.379} C_VEL
LIN {X 0,Y 752.78,Z 954.812,A -85,B 0,C 180,E1 33001.759,E2 33001.759} C_VEL
LIN {X 0,Y 752.838,Z 933.111,A -85,B 0,C 180,E1 33001.34,E2 33001.34} C_VEL
LIN {X 0,Y 752.884,Z 912.621,A -85,B 0,C 180,E1 33001.044,E2 33001.044} C_VEL
LIN {X 0,Y 753.034,Z 654.761,A -85,B 0,C 180,E1 32998.249,E2 32998.249} C_VEL
LIN {X 0,Y 753.009,Z 528.808,A -85,B 0,C 180,E1 32996.85,E2 32996.85} C_VEL
LIN {X 0,Y 752.832,Z 524.865,A -85,B 0,C 180,E1 32996.66,E2 32996.66} C_VEL
LIN {X 0,Y 752.956,Z 482.689,A -85,B 0,C 180,E1 32994.261,E2 32994.261} C_VEL
LIN {X 0,Y 751.945,Z 479.775,A -85,B 0,C 180,E1 32994.004,E2 32994.004} C_VEL
LIN {X 0,Y 751.912,Z 479.563,A -85,B 0,C 180,E1 32991.56,E2 32991.56} C_VEL
LIN {X 0,Y 751.975,Z 479.558,A -85,B 0,C 180,E1 32988.817,E2 32988.817} C_VEL
LIN {X 0,Y 751.929,Z 479.564,A -85,B 0,C 180,E1 32985.896,E2 32985.896} C_VEL
LIN {X 0,Y 751.914,Z 479.558,A -85,B 0,C 180,E1 32983.328,E2 32983.328} C_VEL
LIN {X 0,Y 751.977,Z 479.557,A -85,B 0,C 180,E1 32980.558,E2 32980.558} C_VEL
LIN {X 0,Y 751.928,Z 479.563,A -85,B 0,C 180,E1 32977.616,E2 32977.616} C_VEL
LIN {X 0,Y 751.922,Z 479.558,A -85,B 0,C 180,E1 32974.969,E2 32974.969} C_VEL
LIN {X 0,Y 751.972,Z 479.557,A -85,B 0,C 180,E1 32972.133,E2 32972.133} C_VEL
LIN {X 0,Y 751.926,Z 479.562,A -85,B 0,C 180,E1 32969.298,E2 32969.298} C_VEL
LIN {X 0,Y 751.932,Z 479.558,A -85,B 0,C 180,E1 32966.624,E2 32966.624} C_VEL
LIN {X 0,Y 751.975,Z 479.563,A -85,B 0,C 180,E1 32963.676,E2 32963.676} C_VEL
LIN {X 0,Y 751.924,Z 479.561,A -85,B 0,C 180,E1 32960.96,E2 32960.96} C_VEL
LIN {X 0,Y 751.942,Z 479.556,A -85,B 0,C 180,E1 32958.29,E2 32958.29} C_VEL
LIN {X 0,Y 751.969,Z 479.567,A -85,B 0,C 180,E1 32955.265,E2 32955.265} C_VEL
LIN {X 0,Y 751.923,Z 479.559,A -85,B 0,C 180,E1 32952.518,E2 32952.518} C_VEL
LIN {X 0,Y 751.977,Z 479.554,A -85,B 0,C 180,E1 32949.722,E2 32949.722} C_VEL
LIN {X 0,Y 751.947,Z 479.564,A -85,B 0,C 180,E1 32946.797,E2 32946.797} C_VEL
LIN {X 0,Y 751.933,Z 479.556,A -85,B 0,C 180,E1 32944.041,E2 32944.041} C_VEL
LIN {X 0,Y 751.968,Z 479.559,A -85,B 0,C 180,E1 32941.219,E2 32941.219} C_VEL
LIN {X 0,Y 751.937,Z 479.562,A -85,B 0,C 180,E1 32938.4,E2 32938.4} C_VEL
LIN {X 0,Y 751.946,Z 479.555,A -85,B 0,C 180,E1 32935.653,E2 32935.653} C_VEL
LIN {X 0,Y 751.949,Z 479.563,A -85,B 0,C 180,E1 32934.407,E2 32934.407} C_VEL
LIN {X 0,Y 750.922,Z 479.684,A -85,B 0,C 180,E1 32933.82,E2 32933.82} C_VEL
LIN {X 0,Y 744.509,Z 480.49,A -85,B 0,C 180,E1 32932.177,E2 32932.177} C_VEL
LIN {X 0,Y 743.994,Z 480.547,A -85,B 0,C 180,E1 32931.749,E2 32931.749} C_VEL
LIN {X 0,Y 744.028,Z 480.545,A -85,B 0,C 180,E1 32928.92,E2 32928.92} C_VEL
LIN {X 0,Y 744.005,Z 480.55,A -85,B 0,C 180,E1 32926.08,E2 32926.08} C_VEL
LIN {X 0,Y 744.011,Z 480.544,A -85,B 0,C 180,E1 32923.286,E2 32923.286} C_VEL
LIN {X 0,Y 744.037,Z 480.552,A -85,B 0,C 180,E1 32920.287,E2 32920.287} C_VEL
LIN {X 0,Y 743.995,Z 480.547,A -85,B 0,C 180,E1 32917.479,E2 32917.479} C_VEL
LIN {X 0,Y 744.036,Z 480.543,A -85,B 0,C 180,E1 32914.7,E2 32914.7} C_VEL
LIN {X 0,Y 744.021,Z 480.554,A -85,B 0,C 180,E1 32911.767,E2 32911.767} C_VEL
LIN {X 0,Y 744.017,Z 480.543,A -85,B 0,C 180,E1 32908.842,E2 32908.842} C_VEL
LIN {X 0,Y 744.033,Z 480.553,A -85,B 0,C 180,E1 32905.823,E2 32905.823} C_VEL
LIN {X 0,Y 744,Z 480.543,A -85,B 0,C 180,E1 32902.965,E2 32902.965} C_VEL
LIN {X 0,Y 744.025,Z 480.545,A -85,B 0,C 180,E1 32900.131,E2 32900.131} C_VEL
LIN {X 0,Y 744.017,Z 480.55,A -85,B 0,C 180,E1 32897.26,E2 32897.26} C_VEL
LIN {X 0,Y 744.03,Z 480.543,A -85,B 0,C 180,E1 32894.33,E2 32894.33} C_VEL
LIN {X 0,Y 744.039,Z 480.554,A -85,B 0,C 180,E1 32891.286,E2 32891.286} C_VEL
LIN {X 0,Y 744.012,Z 480.549,A -85,B 0,C 180,E1 32888.38,E2 32888.38} C_VEL
LIN {X 0,Y 744.073,Z 480.792,A -85,B 0,C 180,E1 32886.004,E2 32886.004} C_VEL
LIN {X 0,Y 745.915,Z 486.105,A -85,B 0,C 180,E1 32885.543,E2 32885.543} C_VEL
LIN {X 0,Y 745.607,Z 529.622,A -85,B 0,C 180,E1 32882.895,E2 32882.895} C_VEL
LIN {X 0,Y 745.376,Z 576.7,A -85,B 0,C 180,E1 32880.112,E2 32880.112} C_VEL
LIN {X 0,Y 745.103,Z 625.299,A -85,B 0,C 180,E1 32877.318,E2 32877.318} C_VEL
LIN {X 0,Y 745.084,Z 651.834,A -85,B 0,C 180,E1 32875.842,E2 32875.842} C_VEL
LIN {X 0,Y 745.439,Z 656.967,A -85,B 0,C 180,E1 32875.772,E2 32875.772} C_VEL
LIN {X 0,Y 745.14,Z 932.835,A -85,B 0,C 180,E1 32872.923,E2 32872.923} C_VEL
LIN {X 0,Y 745.068,Z 961.601,A -85,B 0,C 180,E1 32872.582,E2 32872.582} C_VEL
LIN {X 0,Y 745.017,Z 982.765,A -85,B 0,C 180,E1 32872.197,E2 32872.197} C_VEL
LIN {X 0,Y 744.903,Z 1003.229,A -85,B 0,C 180,E1 32871.684,E2 32871.684} C_VEL
LIN {X 0,Y 744.788,Z 1024.694,A -85,B 0,C 180,E1 32871.004,E2 32871.004} C_VEL
LIN {X 0,Y 744.691,Z 1044.62,A -85,B 0,C 180,E1 32870.226,E2 32870.226} C_VEL
LIN {X 0,Y 744.556,Z 1063.403,A -85,B 0,C 180,E1 32869.344,E2 32869.344} C_VEL
LIN {X 0,Y 744.426,Z 1082.054,A -85,B 0,C 180,E1 32868.318,E2 32868.318} C_VEL
LIN {X 0,Y 744.332,Z 1099.63,A -85,B 0,C 180,E1 32867.189,E2 32867.189} C_VEL
LIN {X 0,Y 744.219,Z 1116.646,A -85,B 0,C 180,E1 32865.907,E2 32865.907} C_VEL
LIN {X 0,Y 744.133,Z 1131.235,A -85,B 0,C 180,E1 32864.632,E2 32864.632} C_VEL
LIN {X 0,Y 744.047,Z 1145.344,A -85,B 0,C 180,E1 32863.206,E2 32863.206} C_VEL
LIN {X 0,Y 744.004,Z 1157.372,A -85,B 0,C 180,E1 32861.787,E2 32861.787} C_VEL
LIN {X 0,Y 743.967,Z 1168.028,A -85,B 0,C 180,E1 32860.297,E2 32860.297} C_VEL
LIN {X 0,Y 743.943,Z 1177.427,A -85,B 0,C 180,E1 32858.735,E2 32858.735} C_VEL
LIN {X 0,Y 743.929,Z 1185.027,A -85,B 0,C 180,E1 32857.18,E2 32857.18} C_VEL
LIN {X 0,Y 743.907,Z 1191.253,A -85,B 0,C 180,E1 32855.553,E2 32855.553} C_VEL
LIN {X 0,Y 743.912,Z 1195.897,A -85,B 0,C 180,E1 32853.931,E2 32853.931} C_VEL
LIN {X 0,Y 743.912,Z 1198.942,A -85,B 0,C 180,E1 32852.234,E2 32852.234} C_VEL
LIN {X 0,Y 743.902,Z 1200.338,A -85,B 0,C 180,E1 32850.539,E2 32850.539} C_VEL
LIN {X 0,Y 743.91,Z 1200.186,A -85,B 0,C 180,E1 32848.922,E2 32848.922} C_VEL
LIN {X 0,Y 743.912,Z 1198.291,A -85,B 0,C 180,E1 32847.227,E2 32847.227} C_VEL
LIN {X 0,Y 743.918,Z 1194.723,A -85,B 0,C 180,E1 32845.529,E2 32845.529} C_VEL
LIN {X 0,Y 743.918,Z 1189.753,A -85,B 0,C 180,E1 32843.905,E2 32843.905} C_VEL
LIN {X 0,Y 743.916,Z 1182.962,A -85,B 0,C 180,E1 32842.276,E2 32842.276} C_VEL
LIN {X 0,Y 743.949,Z 1174.4,A -85,B 0,C 180,E1 32840.641,E2 32840.641} C_VEL
LIN {X 0,Y 743.973,Z 1164.449,A -85,B 0,C 180,E1 32839.077,E2 32839.077} C_VEL
LIN {X 0,Y 744.022,Z 1152.99,A -85,B 0,C 180,E1 32837.584,E2 32837.584} C_VEL
LIN {X 0,Y 744.079,Z 1140.221,A -85,B 0,C 180,E1 32836.161,E2 32836.161} C_VEL
LIN {X 0,Y 744.161,Z 1126.179,A -85,B 0,C 180,E1 32834.811,E2 32834.811} C_VEL
LIN {X 0,Y 744.253,Z 1110.194,A -85,B 0,C 180,E1 32833.493,E2 32833.493} C_VEL
LIN {X 0,Y 744.354,Z 1093.078,A -85,B 0,C 180,E1 32832.283,E2 32832.283} C_VEL
LIN {X 0,Y 744.487,Z 1074.465,A -85,B 0,C 180,E1 32831.156,E2 32831.156} C_VEL
LIN {X 0,Y 744.62,Z 1055.854,A -85,B 0,C 180,E1 32830.192,E2 32830.192} C_VEL
LIN {X 0,Y 744.72,Z 1036.806,A -85,B 0,C 180,E1 32829.362,E2 32829.362} C_VEL
LIN {X 0,Y 744.848,Z 1016.002,A -85,B 0,C 180,E1 32828.613,E2 32828.613} C_VEL
LIN {X 0,Y 744.963,Z 995.183,A -85,B 0,C 180,E1 32828.006,E2 32828.006} C_VEL
LIN {X 0,Y 745.026,Z 974.144,A -85,B 0,C 180,E1 32827.541,E2 32827.541} C_VEL
LIN {X 0,Y 745.103,Z 951.942,A -85,B 0,C 180,E1 32827.196,E2 32827.196} C_VEL
LIN {X 0,Y 745.421,Z 672.416,A -85,B 0,C 180,E1 32824.299,E2 32824.299} C_VEL
LIN {X 0,Y 745.202,Z 652.579,A -85,B 0,C 180,E1 32824.083,E2 32824.083} C_VEL
LIN {X 0,Y 745.005,Z 650.535,A -85,B 0,C 180,E1 32824.016,E2 32824.016} C_VEL
LIN {X 0,Y 745.243,Z 600.567,A -85,B 0,C 180,E1 32821.179,E2 32821.179} C_VEL
LIN {X 0,Y 745.49,Z 552.831,A -85,B 0,C 180,E1 32818.397,E2 32818.397} C_VEL
LIN {X 0,Y 745.791,Z 505.228,A -85,B 0,C 180,E1 32815.542,E2 32815.542} C_VEL
LIN {X 0,Y 745.729,Z 485.538,A -85,B 0,C 180,E1 32814.321,E2 32814.321} C_VEL
LIN {X 0,Y 744.061,Z 480.773,A -85,B 0,C 180,E1 32813.902,E2 32813.902} C_VEL
LIN {X 0,Y 744.003,Z 480.552,A -85,B 0,C 180,E1 32811.091,E2 32811.091} C_VEL
LIN {X 0,Y 744.025,Z 480.548,A -85,B 0,C 180,E1 32808.302,E2 32808.302} C_VEL
LIN {X 0,Y 744.005,Z 480.546,A -85,B 0,C 180,E1 32805.421,E2 32805.421} C_VEL
LIN {X 0,Y 744.024,Z 480.549,A -85,B 0,C 180,E1 32802.572,E2 32802.572} C_VEL
LIN {X 0,Y 744.025,Z 480.542,A -85,B 0,C 180,E1 32799.469,E2 32799.469} C_VEL
LIN {X 0,Y 744.001,Z 480.547,A -85,B 0,C 180,E1 32796.635,E2 32796.635} C_VEL
LIN {X 0,Y 744.028,Z 480.548,A -85,B 0,C 180,E1 32793.805,E2 32793.805} C_VEL
LIN {X 0,Y 744,Z 480.546,A -85,B 0,C 180,E1 32790.974,E2 32790.974} C_VEL
LIN {X 0,Y 744.019,Z 480.554,A -85,B 0,C 180,E1 32788.146,E2 32788.146} C_VEL
LIN {X 0,Y 744.019,Z 480.544,A -85,B 0,C 180,E1 32785.045,E2 32785.045} C_VEL
LIN {X 0,Y 743.994,Z 480.549,A -85,B 0,C 180,E1 32782.272,E2 32782.272} C_VEL
LIN {X 0,Y 744.03,Z 480.549,A -85,B 0,C 180,E1 32779.468,E2 32779.468} C_VEL
LIN {X 0,Y 744.002,Z 480.545,A -85,B 0,C 180,E1 32776.626,E2 32776.626} C_VEL
LIN {X 0,Y 744.005,Z 480.551,A -85,B 0,C 180,E1 32773.841,E2 32773.841} C_VEL
LIN {X 0,Y 744.036,Z 480.541,A -85,B 0,C 180,E1 32770.844,E2 32770.844} C_VEL
LIN {X 0,Y 743.987,Z 480.549,A -85,B 0,C 180,E1 32768.035,E2 32768.035} C_VEL
LIN {X 0,Y 744.038,Z 480.554,A -85,B 0,C 180,E1 32765.243,E2 32765.243} C_VEL
LIN {X 0,Y 744,Z 480.545,A -85,B 0,C 180,E1 32762.234,E2 32762.234} C_VEL
LIN {X 0,Y 743.993,Z 480.551,A -85,B 0,C 180,E1 32759.538,E2 32759.538} C_VEL
LIN {X 0,Y 744.031,Z 480.547,A -85,B 0,C 180,E1 32756.687,E2 32756.687} C_VEL
LIN {X 0,Y 743.992,Z 480.547,A -85,B 0,C 180,E1 32753.905,E2 32753.905} C_VEL
LIN {X 0,Y 743.999,Z 480.55,A -85,B 0,C 180,E1 32751.187,E2 32751.187} C_VEL
LIN {X 0,Y 744.038,Z 480.542,A -85,B 0,C 180,E1 32748.213,E2 32748.213} C_VEL
LIN {X 0,Y 743.98,Z 480.549,A -85,B 0,C 180,E1 32745.444,E2 32745.444} C_VEL
LIN {X 0,Y 744.02,Z 480.553,A -85,B 0,C 180,E1 32742.722,E2 32742.722} C_VEL
LIN {X 0,Y 744.01,Z 480.544,A -85,B 0,C 180,E1 32739.712,E2 32739.712} C_VEL
LIN {X 0,Y 743.981,Z 480.551,A -85,B 0,C 180,E1 32737.012,E2 32737.012} C_VEL
LIN {X 0,Y 744.036,Z 480.555,A -85,B 0,C 180,E1 32734.274,E2 32734.274} C_VEL
LIN {X 0,Y 743.991,Z 480.546,A -85,B 0,C 180,E1 32731.328,E2 32731.328} C_VEL
LIN {X 0,Y 743.98,Z 480.551,A -85,B 0,C 180,E1 32728.731,E2 32728.731} C_VEL
LIN {X 0,Y 744.036,Z 480.551,A -85,B 0,C 180,E1 32725.917,E2 32725.917} C_VEL
LIN {X 0,Y 743.99,Z 480.547,A -85,B 0,C 180,E1 32723.076,E2 32723.076} C_VEL
LIN {X 0,Y 743.98,Z 480.546,A -85,B 0,C 180,E1 32720.428,E2 32720.428} C_VEL
LIN {X 0,Y 744.035,Z 480.547,A -85,B 0,C 180,E1 32717.575,E2 32717.575} C_VEL
LIN {X 0,Y 743.983,Z 480.549,A -85,B 0,C 180,E1 32714.766,E2 32714.766} C_VEL
LIN {X 0,Y 743.977,Z 480.549,A -85,B 0,C 180,E1 32712.219,E2 32712.219} C_VEL
LIN {X 0,Y 744.035,Z 480.549,A -85,B 0,C 180,E1 32709.4,E2 32709.4} C_VEL
LIN {X 0,Y 743.982,Z 480.568,A -85,B 0,C 180,E1 32706.515,E2 32706.515} C_VEL
LIN {X 0,Y 744.055,Z 481.067,A -85,B 0,C 180,E1 32706.343,E2 32706.343} C_VEL
LIN {X 0,Y 746.024,Z 486.518,A -85,B 0,C 180,E1 32705.899,E2 32705.899} C_VEL
LIN {X 0,Y 745.806,Z 527.982,A -85,B 0,C 180,E1 32703.528,E2 32703.528} C_VEL
LIN {X 0,Y 746.466,Z 532.546,A -85,B 0,C 180,E1 32703.433,E2 32703.433} C_VEL
LIN {X 0,Y 746.039,Z 791.287,A -85,B 0,C 180,E1 32700.577,E2 32700.577} C_VEL
LIN {X 0,Y 745.863,Z 918.724,A -85,B 0,C 180,E1 32699.176,E2 32699.176} C_VEL
LIN {X 0,Y 745.718,Z 944.086,A -85,B 0,C 180,E1 32698.759,E2 32698.759} C_VEL
LIN {X 0,Y 745.622,Z 965.185,A -85,B 0,C 180,E1 32698.283,E2 32698.283} C_VEL
LIN {X 0,Y 745.506,Z 987.923,A -85,B 0,C 180,E1 32697.649,E2 32697.649} C_VEL
LIN {X 0,Y 745.319,Z 1011.265,A -85,B 0,C 180,E1 32696.839,E2 32696.839} C_VEL
LIN {X 0,Y 745.174,Z 1031.901,A -85,B 0,C 180,E1 32695.997,E2 32695.997} C_VEL
LIN {X 0,Y 744.96,Z 1054.937,A -85,B 0,C 180,E1 32694.894,E2 32694.894} C_VEL
LIN {X 0,Y 744.815,Z 1074.171,A -85,B 0,C 180,E1 32693.833,E2 32693.833} C_VEL
LIN {X 0,Y 744.617,Z 1095.244,A -85,B 0,C 180,E1 32692.501,E2 32692.501} C_VEL
LIN {X 0,Y 744.488,Z 1112.82,A -85,B 0,C 180,E1 32691.237,E2 32691.237} C_VEL
LIN {X 0,Y 744.329,Z 1130.611,A -85,B 0,C 180,E1 32689.786,E2 32689.786} C_VEL
LIN {X 0,Y 744.242,Z 1146.502,A -85,B 0,C 180,E1 32688.323,E2 32688.323} C_VEL
LIN {X 0,Y 744.136,Z 1161.805,A -85,B 0,C 180,E1 32686.711,E2 32686.711} C_VEL
LIN {X 0,Y 744.051,Z 1175.179,A -85,B 0,C 180,E1 32685.111,E2 32685.111} C_VEL
LIN {X 0,Y 743.986,Z 1187.948,A -85,B 0,C 180,E1 32683.336,E2 32683.336} C_VEL
LIN {X 0,Y 743.956,Z 1197.566,A -85,B 0,C 180,E1 32681.788,E2 32681.788} C_VEL
LIN {X 0,Y 743.912,Z 1207.471,A -85,B 0,C 180,E1 32679.906,E2 32679.906} C_VEL
LIN {X 0,Y 743.933,Z 1214.511,A -85,B 0,C 180,E1 32678.268,E2 32678.268} C_VEL
LIN {X 0,Y 743.912,Z 1220.761,A -85,B 0,C 180,E1 32676.483,E2 32676.483} C_VEL
LIN {X 0,Y 743.916,Z 1225.495,A -85,B 0,C 180,E1 32674.625,E2 32674.625} C_VEL
LIN {X 0,Y 743.882,Z 1228.346,A -85,B 0,C 180,E1 32673.005,E2 32673.005} C_VEL
LIN {X 0,Y 743.909,Z 1230.195,A -85,B 0,C 180,E1 32671.078,E2 32671.078} C_VEL
LIN {X 0,Y 743.881,Z 1230.328,A -85,B 0,C 180,E1 32669.384,E2 32669.384} C_VEL
LIN {X 0,Y 743.909,Z 1229.163,A -85,B 0,C 180,E1 32667.612,E2 32667.612} C_VEL
LIN {X 0,Y 743.916,Z 1226.288,A -85,B 0,C 180,E1 32665.761,E2 32665.761} C_VEL
LIN {X 0,Y 743.919,Z 1222.482,A -85,B 0,C 180,E1 32664.137,E2 32664.137} C_VEL
LIN {X 0,Y 743.897,Z 1216.638,A -85,B 0,C 180,E1 32662.276,E2 32662.276} C_VEL
LIN {X 0,Y 743.924,Z 1209.602,A -85,B 0,C 180,E1 32660.562,E2 32660.562} C_VEL
LIN {X 0,Y 743.926,Z 1201.927,A -85,B 0,C 180,E1 32658.998,E2 32658.998} C_VEL
LIN {X 0,Y 743.978,Z 1190.874,A -85,B 0,C 180,E1 32657.109,E2 32657.109} C_VEL
LIN {X 0,Y 744.029,Z 1180.535,A -85,B 0,C 180,E1 32655.605,E2 32655.605} C_VEL
LIN {X 0,Y 744.1,Z 1167.211,A -85,B 0,C 180,E1 32653.903,E2 32653.903} C_VEL
LIN {X 0,Y 744.187,Z 1152.849,A -85,B 0,C 180,E1 32652.323,E2 32652.323} C_VEL
LIN {X 0,Y 744.316,Z 1137.108,A -85,B 0,C 180,E1 32650.785,E2 32650.785} C_VEL
LIN {X 0,Y 744.415,Z 1120.335,A -85,B 0,C 180,E1 32649.355,E2 32649.355} C_VEL
LIN {X 0,Y 744.581,Z 1101.884,A -85,B 0,C 180,E1 32647.956,E2 32647.956} C_VEL
LIN {X 0,Y 744.718,Z 1082.775,A -85,B 0,C 180,E1 32646.689,E2 32646.689} C_VEL
LIN {X 0,Y 744.927,Z 1061.57,A -85,B 0,C 180,E1 32645.454,E2 32645.454} C_VEL
LIN {X 0,Y 745.074,Z 1041.476,A -85,B 0,C 180,E1 32644.441,E2 32644.441} C_VEL
LIN {X 0,Y 745.289,Z 1019.208,A -85,B 0,C 180,E1 32643.465,E2 32643.465} C_VEL
LIN {X 0,Y 745.428,Z 997.568,A -85,B 0,C 180,E1 32642.671,E2 32642.671} C_VEL
LIN {X 0,Y 745.55,Z 976.914,A -85,B 0,C 180,E1 32642.027,E2 32642.027} C_VEL
LIN {X 0,Y 745.695,Z 951.987,A -85,B 0,C 180,E1 32641.407,E2 32641.407} C_VEL
LIN {X 0,Y 745.798,Z 931.654,A -85,B 0,C 180,E1 32641.019,E2 32641.019} C_VEL
LIN {X 0,Y 745.883,Z 908.445,A -85,B 0,C 180,E1 32640.693,E2 32640.693} C_VEL
LIN {X 0,Y 746.219,Z 659.087,A -85,B 0,C 180,E1 32637.972,E2 32637.972} C_VEL
LIN {X 0,Y 746.289,Z 530.397,A -85,B 0,C 180,E1 32636.533,E2 32636.533} C_VEL
LIN {X 0,Y 745.767,Z 527.002,A -85,B 0,C 180,E1 32636.424,E2 32636.424} C_VEL
LIN {X 0,Y 746.023,Z 486.227,A -85,B 0,C 180,E1 32634.084,E2 32634.084} C_VEL
LIN {X 0,Y 744,Z 480.737,A -85,B 0,C 180,E1 32633.613,E2 32633.613} C_VEL
LIN {X 0,Y 744.039,Z 480.547,A -85,B 0,C 180,E1 32630.931,E2 32630.931} C_VEL
LIN {X 0,Y 743.991,Z 480.551,A -85,B 0,C 180,E1 32627.99,E2 32627.99} C_VEL
LIN {X 0,Y 743.975,Z 480.55,A -85,B 0,C 180,E1 32625.424,E2 32625.424} C_VEL
LIN {X 0,Y 744.026,Z 480.543,A -85,B 0,C 180,E1 32622.74,E2 32622.74} C_VEL
LIN {X 0,Y 743.996,Z 480.547,A -85,B 0,C 180,E1 32619.762,E2 32619.762} C_VEL
LIN {X 0,Y 743.979,Z 480.549,A -85,B 0,C 180,E1 32617.117,E2 32617.117} C_VEL
LIN {X 0,Y 744.034,Z 480.545,A -85,B 0,C 180,E1 32614.363,E2 32614.363} C_VEL
LIN {X 0,Y 743.991,Z 480.552,A -85,B 0,C 180,E1 32611.419,E2 32611.419} C_VEL
LIN {X 0,Y 743.986,Z 480.546,A -85,B 0,C 180,E1 32608.76,E2 32608.76} C_VEL
LIN {X 0,Y 744.033,Z 480.55,A -85,B 0,C 180,E1 32605.898,E2 32605.898} C_VEL
LIN {X 0,Y 743.988,Z 480.552,A -85,B 0,C 180,E1 32603.106,E2 32603.106} C_VEL
LIN {X 0,Y 743.995,Z 480.545,A -85,B 0,C 180,E1 32600.452,E2 32600.452} C_VEL
LIN {X 0,Y 744.035,Z 480.552,A -85,B 0,C 180,E1 32597.519,E2 32597.519} C_VEL
LIN {X 0,Y 743.985,Z 480.55,A -85,B 0,C 180,E1 32594.715,E2 32594.715} C_VEL
LIN {X 0,Y 744.024,Z 480.542,A -85,B 0,C 180,E1 32591.944,E2 32591.944} C_VEL
LIN {X 0,Y 744.011,Z 480.551,A -85,B 0,C 180,E1 32588.891,E2 32588.891} C_VEL
LIN {X 0,Y 743.991,Z 480.547,A -85,B 0,C 180,E1 32586.172,E2 32586.172} C_VEL
LIN {X 0,Y 744.031,Z 480.545,A -85,B 0,C 180,E1 32583.39,E2 32583.39} C_VEL
LIN {X 0,Y 743.998,Z 480.551,A -85,B 0,C 180,E1 32580.462,E2 32580.462} C_VEL
LIN {X 0,Y 744.01,Z 480.544,A -85,B 0,C 180,E1 32577.689,E2 32577.689} C_VEL
LIN {X 0,Y 744.034,Z 480.554,A -85,B 0,C 180,E1 32574.679,E2 32574.679} C_VEL
LIN {X 0,Y 743.992,Z 480.548,A -85,B 0,C 180,E1 32571.888,E2 32571.888} C_VEL
LIN {X 0,Y 743.994,Z 480.547,A -85,B 0,C 180,E1 32571.749,E2 32571.749} C_VEL
LIN {X 0,Y 743.03,Z 480.67,A -85,B 0,C 180,E1 32571.156,E2 32571.156} C_VEL
LIN {X 0,Y 736.634,Z 481.463,A -85,B 0,C 180,E1 32569.495,E2 32569.495} C_VEL
LIN {X 0,Y 736.093,Z 481.53,A -85,B 0,C 180,E1 32569.063,E2 32569.063} C_VEL
LIN {X 0,Y 736.068,Z 481.539,A -85,B 0,C 180,E1 32566.087,E2 32566.087} C_VEL
LIN {X 0,Y 736.074,Z 481.533,A -85,B 0,C 180,E1 32563.263,E2 32563.263} C_VEL
LIN {X 0,Y 736.098,Z 481.541,A -85,B 0,C 180,E1 32560.231,E2 32560.231} C_VEL
LIN {X 0,Y 736.058,Z 481.534,A -85,B 0,C 180,E1 32557.391,E2 32557.391} C_VEL
LIN {X 0,Y 736.09,Z 481.535,A -85,B 0,C 180,E1 32554.58,E2 32554.58} C_VEL
LIN {X 0,Y 736.073,Z 481.542,A -85,B 0,C 180,E1 32551.669,E2 32551.669} C_VEL
LIN {X 0,Y 736.088,Z 481.532,A -85,B 0,C 180,E1 32548.741,E2 32548.741} C_VEL
LIN {X 0,Y 736.091,Z 481.544,A -85,B 0,C 180,E1 32545.676,E2 32545.676} C_VEL
LIN {X 0,Y 736.072,Z 481.528,A -85,B 0,C 180,E1 32542.75,E2 32542.75} C_VEL
LIN {X 0,Y 736.086,Z 481.539,A -85,B 0,C 180,E1 32539.817,E2 32539.817} C_VEL
LIN {X 0,Y 736.064,Z 481.536,A -85,B 0,C 180,E1 32537.005,E2 32537.005} C_VEL
LIN {X 0,Y 736.098,Z 481.532,A -85,B 0,C 180,E1 32534.172,E2 32534.172} C_VEL
LIN {X 0,Y 736.082,Z 481.543,A -85,B 0,C 180,E1 32531.105,E2 32531.105} C_VEL
LIN {X 0,Y 736.091,Z 481.537,A -85,B 0,C 180,E1 32528.14,E2 32528.14} C_VEL
LIN {X 0,Y 736.09,Z 481.697,A -85,B 0,C 180,E1 32526.412,E2 32526.412} C_VEL
LIN {X 0,Y 738.147,Z 487.353,A -85,B 0,C 180,E1 32525.899,E2 32525.899} C_VEL
LIN {X 0,Y 738.923,Z 490.198,A -85,B 0,C 180,E1 32525.676,E2 32525.676} C_VEL
LIN {X 0,Y 738.474,Z 534.188,A -85,B 0,C 180,E1 32522.976,E2 32522.976} C_VEL
LIN {X 0,Y 738.096,Z 580.805,A -85,B 0,C 180,E1 32520.198,E2 32520.198} C_VEL
LIN {X 0,Y 737.707,Z 628.347,A -85,B 0,C 180,E1 32517.44,E2 32517.44} C_VEL
LIN {X 0,Y 737.647,Z 651.772,A -85,B 0,C 180,E1 32516.124,E2 32516.124} C_VEL
LIN {X 0,Y 738.234,Z 657.017,A -85,B 0,C 180,E1 32516.042,E2 32516.042} C_VEL
LIN {X 0,Y 737.771,Z 933.013,A -85,B 0,C 180,E1 32513.164,E2 32513.164} C_VEL
LIN {X 0,Y 737.668,Z 961.735,A -85,B 0,C 180,E1 32512.82,E2 32512.82} C_VEL
LIN {X 0,Y 737.584,Z 983.193,A -85,B 0,C 180,E1 32512.424,E2 32512.424} C_VEL
LIN {X 0,Y 737.417,Z 1004.059,A -85,B 0,C 180,E1 32511.893,E2 32511.893} C_VEL
LIN {X 0,Y 737.235,Z 1025.831,A -85,B 0,C 180,E1 32511.188,E2 32511.188} C_VEL
LIN {X 0,Y 737.08,Z 1046.055,A -85,B 0,C 180,E1 32510.383,E2 32510.383} C_VEL
LIN {X 0,Y 736.88,Z 1065.276,A -85,B 0,C 180,E1 32509.458,E2 32509.458} C_VEL
LIN {X 0,Y 736.68,Z 1083.981,A -85,B 0,C 180,E1 32508.399,E2 32508.399} C_VEL
LIN {X 0,Y 736.515,Z 1101.868,A -85,B 0,C 180,E1 32507.214,E2 32507.214} C_VEL
LIN {X 0,Y 736.366,Z 1118.65,A -85,B 0,C 180,E1 32505.919,E2 32505.919} C_VEL
LIN {X 0,Y 736.232,Z 1133.785,A -85,B 0,C 180,E1 32504.551,E2 32504.551} C_VEL
LIN {X 0,Y 736.112,Z 1147.47,A -85,B 0,C 180,E1 32503.11,E2 32503.11} C_VEL
LIN {X 0,Y 736.032,Z 1159.756,A -85,B 0,C 180,E1 32501.598,E2 32501.598} C_VEL
LIN {X 0,Y 735.983,Z 1170.1,A -85,B 0,C 180,E1 32500.093,E2 32500.093} C_VEL
LIN {X 0,Y 735.952,Z 1179.29,A -85,B 0,C 180,E1 32498.47,E2 32498.47} C_VEL
LIN {X 0,Y 735.914,Z 1186.985,A -85,B 0,C 180,E1 32496.788,E2 32496.788} C_VEL
LIN {X 0,Y 735.922,Z 1192.773,A -85,B 0,C 180,E1 32495.145,E2 32495.145} C_VEL
LIN {X 0,Y 735.913,Z 1196.849,A -85,B 0,C 180,E1 32493.505,E2 32493.505} C_VEL
LIN {X 0,Y 735.916,Z 1199.51,A -85,B 0,C 180,E1 32491.791,E2 32491.791} C_VEL
LIN {X 0,Y 735.913,Z 1200.471,A -85,B 0,C 180,E1 32490.078,E2 32490.078} C_VEL
LIN {X 0,Y 735.901,Z 1199.787,A -85,B 0,C 180,E1 32488.443,E2 32488.443} C_VEL
LIN {X 0,Y 735.904,Z 1197.503,A -85,B 0,C 180,E1 32486.729,E2 32486.729} C_VEL
LIN {X 0,Y 735.905,Z 1193.699,A -85,B 0,C 180,E1 32485.09,E2 32485.09} C_VEL
LIN {X 0,Y 735.914,Z 1188.24,A -85,B 0,C 180,E1 32483.447,E2 32483.447} C_VEL
LIN {X 0,Y 735.952,Z 1181.142,A -85,B 0,C 180,E1 32481.799,E2 32481.799} C_VEL
LIN {X 0,Y 735.974,Z 1172.554,A -85,B 0,C 180,E1 32480.223,E2 32480.223} C_VEL
LIN {X 0,Y 736.03,Z 1162.142,A -85,B 0,C 180,E1 32478.64,E2 32478.64} C_VEL
LIN {X 0,Y 736.111,Z 1150.369,A -85,B 0,C 180,E1 32477.129,E2 32477.129} C_VEL
LIN {X 0,Y 736.2,Z 1137.117,A -85,B 0,C 180,E1 32475.689,E2 32475.689} C_VEL
LIN {X 0,Y 736.314,Z 1122.463,A -85,B 0,C 180,E1 32474.322,E2 32474.322} C_VEL
LIN {X 0,Y 736.473,Z 1105.853,A -85,B 0,C 180,E1 32472.988,E2 32472.988} C_VEL
LIN {X 0,Y 736.653,Z 1088.808,A -85,B 0,C 180,E1 32471.809,E2 32471.809} C_VEL
LIN {X 0,Y 736.829,Z 1070.279,A -85,B 0,C 180,E1 32470.717,E2 32470.717} C_VEL
LIN {X 0,Y 737.008,Z 1051.154,A -85,B 0,C 180,E1 32469.761,E2 32469.761} C_VEL
LIN {X 0,Y 737.213,Z 1030.496,A -85,B 0,C 180,E1 32468.894,E2 32468.894} C_VEL
LIN {X 0,Y 737.382,Z 1010.008,A -85,B 0,C 180,E1 32468.19,E2 32468.19} C_VEL
LIN {X 0,Y 737.529,Z 988.752,A -85,B 0,C 180,E1 32467.617,E2 32467.617} C_VEL
LIN {X 0,Y 737.658,Z 965.932,A -85,B 0,C 180,E1 32467.158,E2 32467.158} C_VEL
LIN {X 0,Y 737.75,Z 944.237,A -85,B 0,C 180,E1 32466.862,E2 32466.862} C_VEL
LIN {X 0,Y 738.21,Z 669.946,A -85,B 0,C 180,E1 32464.004,E2 32464.004} C_VEL
LIN {X 0,Y 738.013,Z 653.892,A -85,B 0,C 180,E1 32463.826,E2 32463.826} C_VEL
LIN {X 0,Y 737.596,Z 651.323,A -85,B 0,C 180,E1 32463.774,E2 32463.774} C_VEL
LIN {X 0,Y 737.937,Z 601.03,A -85,B 0,C 180,E1 32460.894,E2 32460.894} C_VEL
LIN {X 0,Y 738.306,Z 553.909,A -85,B 0,C 180,E1 32458.119,E2 32458.119} C_VEL
LIN {X 0,Y 738.773,Z 505.292,A -85,B 0,C 180,E1 32455.171,E2 32455.171} C_VEL
LIN {X 0,Y 738.842,Z 489.078,A -85,B 0,C 180,E1 32454.159,E2 32454.159} C_VEL
LIN {X 0,Y 736.086,Z 481.726,A -85,B 0,C 180,E1 32453.504,E2 32453.504} C_VEL
LIN {X 0,Y 736.095,Z 481.532,A -85,B 0,C 180,E1 32450.73,E2 32450.73} C_VEL
LIN {X 0,Y 736.08,Z 481.53,A -85,B 0,C 180,E1 32447.643,E2 32447.643} C_VEL
LIN {X 0,Y 736.077,Z 481.543,A -85,B 0,C 180,E1 32444.721,E2 32444.721} C_VEL
LIN {X 0,Y 736.1,Z 481.53,A -85,B 0,C 180,E1 32441.663,E2 32441.663} C_VEL
LIN {X 0,Y 736.056,Z 481.538,A -85,B 0,C 180,E1 32438.874,E2 32438.874} C_VEL
LIN {X 0,Y 736.092,Z 481.541,A -85,B 0,C 180,E1 32436.028,E2 32436.028} C_VEL
LIN {X 0,Y 736.066,Z 481.533,A -85,B 0,C 180,E1 32433.099,E2 32433.099} C_VEL
LIN {X 0,Y 736.079,Z 481.542,A -85,B 0,C 180,E1 32430.241,E2 32430.241} C_VEL
LIN {X 0,Y 736.09,Z 481.53,A -85,B 0,C 180,E1 32427.156,E2 32427.156} C_VEL
LIN {X 0,Y 736.058,Z 481.54,A -85,B 0,C 180,E1 32424.306,E2 32424.306} C_VEL
LIN {X 0,Y 736.09,Z 481.538,A -85,B 0,C 180,E1 32421.433,E2 32421.433} C_VEL
LIN {X 0,Y 736.059,Z 481.533,A -85,B 0,C 180,E1 32418.617,E2 32418.617} C_VEL
LIN {X 0,Y 736.072,Z 481.542,A -85,B 0,C 180,E1 32415.845,E2 32415.845} C_VEL
LIN {X 0,Y 736.088,Z 481.532,A -85,B 0,C 180,E1 32412.765,E2 32412.765} C_VEL
LIN {X 0,Y 736.05,Z 481.536,A -85,B 0,C 180,E1 32409.988,E2 32409.988} C_VEL
LIN {X 0,Y 736.094,Z 481.539,A -85,B 0,C 180,E1 32407.179,E2 32407.179} C_VEL
LIN {X 0,Y 736.062,Z 481.534,A -85,B 0,C 180,E1 32404.285,E2 32404.285} C_VEL
LIN {X 0,Y 736.056,Z 481.54,A -85,B 0,C 180,E1 32401.557,E2 32401.557} C_VEL
LIN {X 0,Y 736.095,Z 481.535,A -85,B 0,C 180,E1 32398.659,E2 32398.659} C_VEL
LIN {X 0,Y 736.049,Z 481.534,A -85,B 0,C 180,E1 32395.871,E2 32395.871} C_VEL
LIN {X 0,Y 736.072,Z 481.543,A -85,B 0,C 180,E1 32393.134,E2 32393.134} C_VEL
LIN {X 0,Y 736.072,Z 481.534,A -85,B 0,C 180,E1 32390.003,E2 32390.003} C_VEL
LIN {X 0,Y 736.047,Z 481.538,A -85,B 0,C 180,E1 32387.249,E2 32387.249} C_VEL
LIN {X 0,Y 736.095,Z 481.537,A -85,B 0,C 180,E1 32384.376,E2 32384.376} C_VEL
LIN {X 0,Y 736.051,Z 481.536,A -85,B 0,C 180,E1 32381.547,E2 32381.547} C_VEL
LIN {X 0,Y 736.051,Z 481.539,A -85,B 0,C 180,E1 32378.9,E2 32378.9} C_VEL
LIN {X 0,Y 736.095,Z 481.535,A -85,B 0,C 180,E1 32376.036,E2 32376.036} C_VEL
LIN {X 0,Y 736.044,Z 481.537,A -85,B 0,C 180,E1 32373.187,E2 32373.187} C_VEL
LIN {X 0,Y 736.059,Z 481.541,A -85,B 0,C 180,E1 32370.543,E2 32370.543} C_VEL
LIN {X 0,Y 736.086,Z 481.527,A -85,B 0,C 180,E1 32367.515,E2 32367.515} C_VEL
LIN {X 0,Y 736.038,Z 481.537,A -85,B 0,C 180,E1 32364.831,E2 32364.831} C_VEL
LIN {X 0,Y 736.078,Z 481.544,A -85,B 0,C 180,E1 32362.111,E2 32362.111} C_VEL
LIN {X 0,Y 736.059,Z 481.537,A -85,B 0,C 180,E1 32359.049,E2 32359.049} C_VEL
LIN {X 0,Y 736.037,Z 481.536,A -85,B 0,C 180,E1 32356.389,E2 32356.389} C_VEL
LIN {X 0,Y 736.099,Z 481.539,A -85,B 0,C 180,E1 32353.613,E2 32353.613} C_VEL
LIN {X 0,Y 736.046,Z 481.54,A -85,B 0,C 180,E1 32350.695,E2 32350.695} C_VEL
LIN {X 0,Y 736.038,Z 481.546,A -85,B 0,C 180,E1 32348.077,E2 32348.077} C_VEL
LIN {X 0,Y 736.099,Z 481.783,A -85,B 0,C 180,E1 32346.773,E2 32346.773} C_VEL
LIN {X 0,Y 739.086,Z 489.987,A -85,B 0,C 180,E1 32346.084,E2 32346.084} C_VEL
LIN {X 0,Y 738.776,Z 528.02,A -85,B 0,C 180,E1 32343.89,E2 32343.89} C_VEL
LIN {X 0,Y 739.779,Z 534.025,A -85,B 0,C 180,E1 32343.759,E2 32343.759} C_VEL
LIN {X 0,Y 739.143,Z 792.305,A -85,B 0,C 180,E1 32340.882,E2 32340.882} C_VEL
LIN {X 0,Y 738.867,Z 918.831,A -85,B 0,C 180,E1 32339.478,E2 32339.478} C_VEL
LIN {X 0,Y 738.661,Z 944.236,A -85,B 0,C 180,E1 32339.056,E2 32339.056} C_VEL
LIN {X 0,Y 738.509,Z 965.619,A -85,B 0,C 180,E1 32338.569,E2 32338.569} C_VEL
LIN {X 0,Y 738.329,Z 988.653,A -85,B 0,C 180,E1 32337.919,E2 32337.919} C_VEL
LIN {X 0,Y 738.045,Z 1011.538,A -85,B 0,C 180,E1 32337.115,E2 32337.115} C_VEL
LIN {X 0,Y 737.827,Z 1032.256,A -85,B 0,C 180,E1 32336.26,E2 32336.26} C_VEL
LIN {X 0,Y 737.504,Z 1055.157,A -85,B 0,C 180,E1 32335.152,E2 32335.152} C_VEL
LIN {X 0,Y 737.279,Z 1074.901,A -85,B 0,C 180,E1 32334.049,E2 32334.049} C_VEL
LIN {X 0,Y 736.987,Z 1095.246,A -85,B 0,C 180,E1 32332.746,E2 32332.746} C_VEL
LIN {X 0,Y 736.791,Z 1113.062,A -85,B 0,C 180,E1 32331.452,E2 32331.452} C_VEL
LIN {X 0,Y 736.562,Z 1130.611,A -85,B 0,C 180,E1 32330.004,E2 32330.004} C_VEL
LIN {X 0,Y 736.424,Z 1146.501,A -85,B 0,C 180,E1 32328.524,E2 32328.524} C_VEL
LIN {X 0,Y 736.245,Z 1161.807,A -85,B 0,C 180,E1 32326.895,E2 32326.895} C_VEL
LIN {X 0,Y 736.139,Z 1174.717,A -85,B 0,C 180,E1 32325.336,E2 32325.336} C_VEL
LIN {X 0,Y 736.044,Z 1187.757,A -85,B 0,C 180,E1 32323.512,E2 32323.512} C_VEL
LIN {X 0,Y 735.986,Z 1197.133,A -85,B 0,C 180,E1 32321.992,E2 32321.992} C_VEL
LIN {X 0,Y 735.947,Z 1206.762,A -85,B 0,C 180,E1 32320.173,E2 32320.173} C_VEL
LIN {X 0,Y 735.928,Z 1214.208,A -85,B 0,C 180,E1 32318.438,E2 32318.438} C_VEL
LIN {X 0,Y 735.919,Z 1219.998,A -85,B 0,C 180,E1 32316.788,E2 32316.788} C_VEL
LIN {X 0,Y 735.898,Z 1225.178,A -85,B 0,C 180,E1 32314.832,E2 32314.832} C_VEL
LIN {X 0,Y 735.892,Z 1228.122,A -85,B 0,C 180,E1 32313.193,E2 32313.193} C_VEL
LIN {X 0,Y 735.904,Z 1230.099,A -85,B 0,C 180,E1 32311.324,E2 32311.324} C_VEL
LIN {X 0,Y 735.881,Z 1230.351,A -85,B 0,C 180,E1 32309.455,E2 32309.455} C_VEL
LIN {X 0,Y 735.918,Z 1229.297,A -85,B 0,C 180,E1 32307.742,E2 32307.742} C_VEL
LIN {X 0,Y 735.915,Z 1226.288,A -85,B 0,C 180,E1 32305.715,E2 32305.715} C_VEL
LIN {X 0,Y 735.921,Z 1222.357,A -85,B 0,C 180,E1 32304.026,E2 32304.026} C_VEL
LIN {X 0,Y 735.915,Z 1216.271,A -85,B 0,C 180,E1 32302.096,E2 32302.096} C_VEL
LIN {X 0,Y 735.926,Z 1209.247,A -85,B 0,C 180,E1 32300.38,E2 32300.38} C_VEL
LIN {X 0,Y 735.965,Z 1201.113,A -85,B 0,C 180,E1 32298.718,E2 32298.718} C_VEL
LIN {X 0,Y 736.02,Z 1190.356,A -85,B 0,C 180,E1 32296.888,E2 32296.888} C_VEL
LIN {X 0,Y 736.108,Z 1179.958,A -85,B 0,C 180,E1 32295.366,E2 32295.366} C_VEL
LIN {X 0,Y 736.219,Z 1166.05,A -85,B 0,C 180,E1 32293.592,E2 32293.592} C_VEL
LIN {X 0,Y 736.329,Z 1152.074,A -85,B 0,C 180,E1 32292.047,E2 32292.047} C_VEL
LIN {X 0,Y 736.53,Z 1135.255,A -85,B 0,C 180,E1 32290.409,E2 32290.409} C_VEL
LIN {X 0,Y 736.711,Z 1118.815,A -85,B 0,C 180,E1 32289.004,E2 32289.004} C_VEL
LIN {X 0,Y 736.964,Z 1098.867,A -85,B 0,C 180,E1 32287.505,E2 32287.505} C_VEL
LIN {X 0,Y 737.195,Z 1080.356,A -85,B 0,C 180,E1 32286.282,E2 32286.282} C_VEL
LIN {X 0,Y 737.479,Z 1058.364,A -85,B 0,C 180,E1 32285.019,E2 32285.019} C_VEL
LIN {X 0,Y 737.719,Z 1038.809,A -85,B 0,C 180,E1 32284.038,E2 32284.038} C_VEL
LIN {X 0,Y 738.022,Z 1015.4,A -85,B 0,C 180,E1 32283.035,E2 32283.035} C_VEL
LIN {X 0,Y 738.216,Z 995.727,A -85,B 0,C 180,E1 32282.318,E2 32282.318} C_VEL
LIN {X 0,Y 738.492,Z 972.084,A -85,B 0,C 180,E1 32281.596,E2 32281.596} C_VEL
LIN {X 0,Y 738.638,Z 949.369,A -85,B 0,C 180,E1 32281.052,E2 32281.052} C_VEL
LIN {X 0,Y 738.791,Z 928.283,A -85,B 0,C 180,E1 32280.66,E2 32280.66} C_VEL
LIN {X 0,Y 738.935,Z 897.275,A -85,B 0,C 180,E1 32280.266,E2 32280.266} C_VEL
LIN {X 0,Y 739.444,Z 652.521,A -85,B 0,C 180,E1 32277.57,E2 32277.57} C_VEL
LIN {X 0,Y 739.615,Z 532.113,A -85,B 0,C 180,E1 32276.211,E2 32276.211} C_VEL
LIN {X 0,Y 738.734,Z 527.152,A -85,B 0,C 180,E1 32276.069,E2 32276.069} C_VEL
LIN {X 0,Y 739.005,Z 489.407,A -85,B 0,C 180,E1 32273.878,E2 32273.878} C_VEL
LIN {X 0,Y 736.099,Z 481.782,A -85,B 0,C 180,E1 32273.227,E2 32273.227} C_VEL
LIN {X 0,Y 736.095,Z 481.538,A -85,B 0,C 180,E1 32270.427,E2 32270.427} C_VEL
LIN {X 0,Y 736.035,Z 481.536,A -85,B 0,C 180,E1 32267.648,E2 32267.648} C_VEL
LIN {X 0,Y 736.072,Z 481.536,A -85,B 0,C 180,E1 32264.951,E2 32264.951} C_VEL
LIN {X 0,Y 736.064,Z 481.544,A -85,B 0,C 180,E1 32261.893,E2 32261.893} C_VEL
LIN {X 0,Y 736.037,Z 481.53,A -85,B 0,C 180,E1 32259.258,E2 32259.258} C_VEL
LIN {X 0,Y 736.096,Z 481.535,A -85,B 0,C 180,E1 32256.474,E2 32256.474} C_VEL
LIN {X 0,Y 736.051,Z 481.535,A -85,B 0,C 180,E1 32253.482,E2 32253.482} C_VEL
LIN {X 0,Y 736.049,Z 481.536,A -85,B 0,C 180,E1 32250.807,E2 32250.807} C_VEL
LIN {X 0,Y 736.096,Z 481.54,A -85,B 0,C 180,E1 32247.858,E2 32247.858} C_VEL
LIN {X 0,Y 736.044,Z 481.537,A -85,B 0,C 180,E1 32245.033,E2 32245.033} C_VEL
LIN {X 0,Y 736.073,Z 481.534,A -85,B 0,C 180,E1 32242.325,E2 32242.325} C_VEL
LIN {X 0,Y 736.076,Z 481.543,A -85,B 0,C 180,E1 32239.255,E2 32239.255} C_VEL
LIN {X 0,Y 736.048,Z 481.535,A -85,B 0,C 180,E1 32236.494,E2 32236.494} C_VEL
LIN {X 0,Y 736.094,Z 481.536,A -85,B 0,C 180,E1 32233.672,E2 32233.672} C_VEL
LIN {X 0,Y 736.059,Z 481.541,A -85,B 0,C 180,E1 32230.805,E2 32230.805} C_VEL
LIN {X 0,Y 736.066,Z 481.531,A -85,B 0,C 180,E1 32228.005,E2 32228.005} C_VEL
LIN {X 0,Y 736.095,Z 481.543,A -85,B 0,C 180,E1 32224.987,E2 32224.987} C_VEL
LIN {X 0,Y 736.049,Z 481.537,A -85,B 0,C 180,E1 32222.18,E2 32222.18} C_VEL
LIN {X 0,Y 736.095,Z 481.532,A -85,B 0,C 180,E1 32219.377,E2 32219.377} C_VEL
LIN {X 0,Y 736.066,Z 481.541,A -85,B 0,C 180,E1 32216.417,E2 32216.417} C_VEL
LIN {X 0,Y 736.068,Z 481.532,A -85,B 0,C 180,E1 32213.604,E2 32213.604} C_VEL
LIN {X 0,Y 736.097,Z 481.543,A -85,B 0,C 180,E1 32210.619,E2 32210.619} C_VEL
LIN {X 0,Y 736.093,Z 481.53,A -85,B 0,C 180,E1 32209.063,E2 32209.063} C_VEL
LIN {X 0,Y 735.1,Z 481.666,A -85,B 0,C 180,E1 32208.464,E2 32208.464} C_VEL
LIN {X 0,Y 728.697,Z 482.471,A -85,B 0,C 180,E1 32206.785,E2 32206.785} C_VEL
LIN {X 0,Y 728.153,Z 482.53,A -85,B 0,C 180,E1 32206.349,E2 32206.349} C_VEL
LIN {X 0,Y 728.121,Z 482.525,A -85,B 0,C 180,E1 32203.485,E2 32203.485} C_VEL
LIN {X 0,Y 728.15,Z 482.523,A -85,B 0,C 180,E1 32200.622,E2 32200.622} C_VEL
LIN {X 0,Y 728.125,Z 482.526,A -85,B 0,C 180,E1 32197.749,E2 32197.749} C_VEL
LIN {X 0,Y 728.149,Z 482.521,A -85,B 0,C 180,E1 32194.892,E2 32194.892} C_VEL
LIN {X 0,Y 728.147,Z 482.532,A -85,B 0,C 180,E1 32191.811,E2 32191.811} C_VEL
LIN {X 0,Y 728.134,Z 482.523,A -85,B 0,C 180,E1 32188.913,E2 32188.913} C_VEL
LIN {X 0,Y 728.152,Z 482.529,A -85,B 0,C 180,E1 32185.926,E2 32185.926} C_VEL
LIN {X 0,Y 728.122,Z 482.519,A -85,B 0,C 180,E1 32183.054,E2 32183.054} C_VEL
LIN {X 0,Y 728.151,Z 482.522,A -85,B 0,C 180,E1 32180.215,E2 32180.215} C_VEL
LIN {X 0,Y 728.141,Z 482.523,A -85,B 0,C 180,E1 32177.277,E2 32177.277} C_VEL
LIN {X 0,Y 728.152,Z 482.522,A -85,B 0,C 180,E1 32174.321,E2 32174.321} C_VEL
LIN {X 0,Y 728.153,Z 482.533,A -85,B 0,C 180,E1 32171.192,E2 32171.192} C_VEL
LIN {X 0,Y 728.151,Z 482.528,A -85,B 0,C 180,E1 32168.164,E2 32168.164} C_VEL
LIN {X 0,Y 728.164,Z 482.761,A -85,B 0,C 180,E1 32166.797,E2 32166.797} C_VEL
LIN {X 0,Y 731.949,Z 492.946,A -85,B 0,C 180,E1 32165.896,E2 32165.896} C_VEL
LIN {X 0,Y 731.351,Z 537.236,A -85,B 0,C 180,E1 32163.151,E2 32163.151} C_VEL
LIN {X 0,Y 730.831,Z 583.554,A -85,B 0,C 180,E1 32160.366,E2 32160.366} C_VEL
LIN {X 0,Y 730.313,Z 631.394,A -85,B 0,C 180,E1 32157.565,E2 32157.565} C_VEL
LIN {X 0,Y 730.191,Z 651.431,A -85,B 0,C 180,E1 32156.419,E2 32156.419} C_VEL
LIN {X 0,Y 731.043,Z 658.05,A -85,B 0,C 180,E1 32156.307,E2 32156.307} C_VEL
LIN {X 0,Y 730.414,Z 933.7,A -85,B 0,C 180,E1 32153.404,E2 32153.404} C_VEL
LIN {X 0,Y 730.28,Z 962.161,A -85,B 0,C 180,E1 32153.058,E2 32153.058} C_VEL
LIN {X 0,Y 730.159,Z 983.766,A -85,B 0,C 180,E1 32152.653,E2 32152.653} C_VEL
LIN {X 0,Y 729.94,Z 1004.815,A -85,B 0,C 180,E1 32152.108,E2 32152.108} C_VEL
LIN {X 0,Y 729.703,Z 1025.845,A -85,B 0,C 180,E1 32151.418,E2 32151.418} C_VEL
LIN {X 0,Y 729.497,Z 1045.622,A -85,B 0,C 180,E1 32150.625,E2 32150.625} C_VEL
LIN {X 0,Y 729.221,Z 1065.289,A -85,B 0,C 180,E1 32149.671,E2 32149.671} C_VEL
LIN {X 0,Y 728.952,Z 1084.203,A -85,B 0,C 180,E1 32148.588,E2 32148.588} C_VEL
LIN {X 0,Y 728.733,Z 1101.873,A -85,B 0,C 180,E1 32147.404,E2 32147.404} C_VEL
LIN {X 0,Y 728.53,Z 1118.656,A -85,B 0,C 180,E1 32146.095,E2 32146.095} C_VEL
LIN {X 0,Y 728.348,Z 1133.789,A -85,B 0,C 180,E1 32144.712,E2 32144.712} C_VEL
LIN {X 0,Y 728.187,Z 1147.471,A -85,B 0,C 180,E1 32143.256,E2 32143.256} C_VEL
LIN {X 0,Y 728.08,Z 1159.879,A -85,B 0,C 180,E1 32141.71,E2 32141.71} C_VEL
LIN {X 0,Y 728.01,Z 1170.617,A -85,B 0,C 180,E1 32140.125,E2 32140.125} C_VEL
LIN {X 0,Y 727.964,Z 1179.504,A -85,B 0,C 180,E1 32138.523,E2 32138.523} C_VEL
LIN {X 0,Y 727.918,Z 1187.29,A -85,B 0,C 180,E1 32136.784,E2 32136.784} C_VEL
LIN {X 0,Y 727.922,Z 1193.028,A -85,B 0,C 180,E1 32135.122,E2 32135.122} C_VEL
LIN {X 0,Y 727.912,Z 1197.008,A -85,B 0,C 180,E1 32133.465,E2 32133.465} C_VEL
LIN {X 0,Y 727.911,Z 1199.644,A -85,B 0,C 180,E1 32131.653,E2 32131.653} C_VEL
LIN {X 0,Y 727.915,Z 1200.495,A -85,B 0,C 180,E1 32129.921,E2 32129.921} C_VEL
LIN {X 0,Y 727.916,Z 1199.588,A -85,B 0,C 180,E1 32128.19,E2 32128.19} C_VEL
LIN {X 0,Y 727.912,Z 1197.03,A -85,B 0,C 180,E1 32126.456,E2 32126.456} C_VEL
LIN {X 0,Y 727.919,Z 1193.062,A -85,B 0,C 180,E1 32124.799,E2 32124.799} C_VEL
LIN {X 0,Y 727.917,Z 1187.331,A -85,B 0,C 180,E1 32123.137,E2 32123.137} C_VEL
LIN {X 0,Y 727.959,Z 1179.516,A -85,B 0,C 180,E1 32121.39,E2 32121.39} C_VEL
LIN {X 0,Y 728.014,Z 1170.683,A -85,B 0,C 180,E1 32119.795,E2 32119.795} C_VEL
LIN {X 0,Y 728.071,Z 1160.408,A -85,B 0,C 180,E1 32118.273,E2 32118.273} C_VEL
LIN {X 0,Y 728.184,Z 1148.257,A -85,B 0,C 180,E1 32116.744,E2 32116.744} C_VEL
LIN {X 0,Y 728.342,Z 1134.725,A -85,B 0,C 180,E1 32115.288,E2 32115.288} C_VEL
LIN {X 0,Y 728.508,Z 1119.596,A -85,B 0,C 180,E1 32113.898,E2 32113.898} C_VEL
LIN {X 0,Y 728.711,Z 1103.088,A -85,B 0,C 180,E1 32112.596,E2 32112.596} C_VEL
LIN {X 0,Y 728.944,Z 1084.835,A -85,B 0,C 180,E1 32111.362,E2 32111.362} C_VEL
LIN {X 0,Y 729.212,Z 1066.221,A -85,B 0,C 180,E1 32110.287,E2 32110.287} C_VEL
LIN {X 0,Y 729.471,Z 1046.918,A -85,B 0,C 180,E1 32109.345,E2 32109.345} C_VEL
LIN {X 0,Y 729.691,Z 1027.125,A -85,B 0,C 180,E1 32108.54,E2 32108.54} C_VEL
LIN {X 0,Y 729.937,Z 1005.473,A -85,B 0,C 180,E1 32107.821,E2 32107.821} C_VEL
LIN {X 0,Y 730.151,Z 984.11,A -85,B 0,C 180,E1 32107.265,E2 32107.265} C_VEL
LIN {X 0,Y 730.279,Z 962.613,A -85,B 0,C 180,E1 32106.86,E2 32106.86} C_VEL
LIN {X 0,Y 730.415,Z 934.363,A -85,B 0,C 180,E1 32106.513,E2 32106.513} C_VEL
LIN {X 0,Y 731.046,Z 656.405,A -85,B 0,C 180,E1 32103.585,E2 32103.585} C_VEL
LIN {X 0,Y 730.188,Z 651.329,A -85,B 0,C 180,E1 32103.487,E2 32103.487} C_VEL
LIN {X 0,Y 730.639,Z 601.781,A -85,B 0,C 180,E1 32100.62,E2 32100.62} C_VEL
LIN {X 0,Y 731.14,Z 555.014,A -85,B 0,C 180,E1 32097.837,E2 32097.837} C_VEL
LIN {X 0,Y 731.777,Z 506.007,A -85,B 0,C 180,E1 32094.832,E2 32094.832} C_VEL
LIN {X 0,Y 731.896,Z 492.41,A -85,B 0,C 180,E1 32093.976,E2 32093.976} C_VEL
LIN {X 0,Y 728.158,Z 482.743,A -85,B 0,C 180,E1 32093.109,E2 32093.109} C_VEL
LIN {X 0,Y 728.147,Z 482.522,A -85,B 0,C 180,E1 32090.319,E2 32090.319} C_VEL
LIN {X 0,Y 728.129,Z 482.52,A -85,B 0,C 180,E1 32087.499,E2 32087.499} C_VEL
LIN {X 0,Y 728.144,Z 482.533,A -85,B 0,C 180,E1 32084.66,E2 32084.66} C_VEL
LIN {X 0,Y 728.149,Z 482.52,A -85,B 0,C 180,E1 32081.549,E2 32081.549} C_VEL
LIN {X 0,Y 728.127,Z 482.529,A -85,B 0,C 180,E1 32078.669,E2 32078.669} C_VEL
LIN {X 0,Y 728.153,Z 482.524,A -85,B 0,C 180,E1 32075.705,E2 32075.705} C_VEL
LIN {X 0,Y 728.117,Z 482.524,A -85,B 0,C 180,E1 32072.85,E2 32072.85} C_VEL
LIN {X 0,Y 728.16,Z 482.53,A -85,B 0,C 180,E1 32069.989,E2 32069.989} C_VEL
LIN {X 0,Y 728.131,Z 482.521,A -85,B 0,C 180,E1 32066.976,E2 32066.976} C_VEL
LIN {X 0,Y 728.129,Z 482.531,A -85,B 0,C 180,E1 32064.156,E2 32064.156} C_VEL
LIN {X 0,Y 728.159,Z 482.522,A -85,B 0,C 180,E1 32061.171,E2 32061.171} C_VEL
LIN {X 0,Y 728.112,Z 482.524,A -85,B 0,C 180,E1 32058.329,E2 32058.329} C_VEL
LIN {X 0,Y 728.157,Z 482.528,A -85,B 0,C 180,E1 32055.532,E2 32055.532} C_VEL
LIN {X 0,Y 728.125,Z 482.524,A -85,B 0,C 180,E1 32052.531,E2 32052.531} C_VEL
LIN {X 0,Y 728.126,Z 482.527,A -85,B 0,C 180,E1 32049.724,E2 32049.724} C_VEL
LIN {X 0,Y 728.156,Z 482.519,A -85,B 0,C 180,E1 32046.703,E2 32046.703} C_VEL
LIN {X 0,Y 728.109,Z 482.527,A -85,B 0,C 180,E1 32043.937,E2 32043.937} C_VEL
LIN {X 0,Y 728.161,Z 482.529,A -85,B 0,C 180,E1 32041.102,E2 32041.102} C_VEL
LIN {X 0,Y 728.122,Z 482.524,A -85,B 0,C 180,E1 32038.111,E2 32038.111} C_VEL
LIN {X 0,Y 728.119,Z 482.528,A -85,B 0,C 180,E1 32035.353,E2 32035.353} C_VEL
LIN {X 0,Y 728.157,Z 482.519,A -85,B 0,C 180,E1 32032.346,E2 32032.346} C_VEL
LIN {X 0,Y 728.106,Z 482.527,A -85,B 0,C 180,E1 32029.556,E2 32029.556} C_VEL
LIN {X 0,Y 728.155,Z 482.529,A -85,B 0,C 180,E1 32026.743,E2 32026.743} C_VEL
LIN {X 0,Y 728.12,Z 482.522,A -85,B 0,C 180,E1 32023.713,E2 32023.713} C_VEL
LIN {X 0,Y 728.111,Z 482.529,A -85,B 0,C 180,E1 32021.006,E2 32021.006} C_VEL
LIN {X 0,Y 728.159,Z 482.525,A -85,B 0,C 180,E1 32018.068,E2 32018.068} C_VEL
LIN {X 0,Y 728.104,Z 482.524,A -85,B 0,C 180,E1 32015.238,E2 32015.238} C_VEL
LIN {X 0,Y 728.13,Z 482.532,A -85,B 0,C 180,E1 32012.508,E2 32012.508} C_VEL
LIN {X 0,Y 728.13,Z 482.524,A -85,B 0,C 180,E1 32009.427,E2 32009.427} C_VEL
LIN {X 0,Y 728.1,Z 482.52,A -85,B 0,C 180,E1 32006.752,E2 32006.752} C_VEL
LIN {X 0,Y 728.161,Z 482.531,A -85,B 0,C 180,E1 32003.907,E2 32003.907} C_VEL
LIN {X 0,Y 728.111,Z 482.515,A -85,B 0,C 180,E1 32001.009,E2 32001.009} C_VEL
LIN {X 0,Y 728.105,Z 482.531,A -85,B 0,C 180,E1 31998.343,E2 31998.343} C_VEL
LIN {X 0,Y 728.158,Z 482.527,A -85,B 0,C 180,E1 31995.437,E2 31995.437} C_VEL
LIN {X 0,Y 728.098,Z 482.523,A -85,B 0,C 180,E1 31992.601,E2 31992.601} C_VEL
LIN {X 0,Y 728.112,Z 482.535,A -85,B 0,C 180,E1 31989.979,E2 31989.979} C_VEL
LIN {X 0,Y 728.192,Z 482.748,A -85,B 0,C 180,E1 31987.184,E2 31987.184} C_VEL
LIN {X 0,Y 730.61,Z 489.136,A -85,B 0,C 180,E1 31986.621,E2 31986.621} C_VEL
LIN {X 0,Y 732.159,Z 493.314,A -85,B 0,C 180,E1 31986.28,E2 31986.28} C_VEL
LIN {X 0,Y 731.818,Z 528.395,A -85,B 0,C 180,E1 31984.247,E2 31984.247} C_VEL
LIN {X 0,Y 733.116,Z 535.541,A -85,B 0,C 180,E1 31984.09,E2 31984.09} C_VEL
LIN {X 0,Y 732.269,Z 793.45,A -85,B 0,C 180,E1 31981.191,E2 31981.191} C_VEL
LIN {X 0,Y 731.891,Z 918.939,A -85,B 0,C 180,E1 31979.786,E2 31979.786} C_VEL
LIN {X 0,Y 731.625,Z 944.561,A -85,B 0,C 180,E1 31979.356,E2 31979.356} C_VEL
LIN {X 0,Y 731.415,Z 965.945,A -85,B 0,C 180,E1 31978.864,E2 31978.864} C_VEL
LIN {X 0,Y 731.159,Z 989.321,A -85,B 0,C 180,E1 31978.195,E2 31978.195} C_VEL
LIN {X 0,Y 730.784,Z 1012.274,A -85,B 0,C 180,E1 31977.378,E2 31977.378} C_VEL
LIN {X 0,Y 730.483,Z 1034.068,A -85,B 0,C 180,E1 31976.465,E2 31976.465} C_VEL
LIN {X 0,Y 730.06,Z 1055.963,A -85,B 0,C 180,E1 31975.383,E2 31975.383} C_VEL
LIN {X 0,Y 729.749,Z 1076.358,A -85,B 0,C 180,E1 31974.227,E2 31974.227} C_VEL
LIN {X 0,Y 729.359,Z 1096.455,A -85,B 0,C 180,E1 31972.913,E2 31972.913} C_VEL
LIN {X 0,Y 729.084,Z 1115.261,A -85,B 0,C 180,E1 31971.521,E2 31971.521} C_VEL
LIN {X 0,Y 728.776,Z 1132.469,A -85,B 0,C 180,E1 31970.059,E2 31970.059} C_VEL
LIN {X 0,Y 728.567,Z 1148.968,A -85,B 0,C 180,E1 31968.482,E2 31968.482} C_VEL
LIN {X 0,Y 728.359,Z 1163.443,A -85,B 0,C 180,E1 31966.894,E2 31966.894} C_VEL
LIN {X 0,Y 728.207,Z 1177.062,A -85,B 0,C 180,E1 31965.204,E2 31965.204} C_VEL
LIN {X 0,Y 728.087,Z 1188.797,A -85,B 0,C 180,E1 31963.501,E2 31963.501} C_VEL
LIN {X 0,Y 728.016,Z 1198.953,A -85,B 0,C 180,E1 31961.808,E2 31961.808} C_VEL
LIN {X 0,Y 727.941,Z 1208.183,A -85,B 0,C 180,E1 31959.966,E2 31959.966} C_VEL
LIN {X 0,Y 727.941,Z 1214.816,A -85,B 0,C 180,E1 31958.372,E2 31958.372} C_VEL
LIN {X 0,Y 727.918,Z 1221.245,A -85,B 0,C 180,E1 31956.467,E2 31956.467} C_VEL
LIN {X 0,Y 727.918,Z 1225.813,A -85,B 0,C 180,E1 31954.569,E2 31954.569} C_VEL
LIN {X 0,Y 727.882,Z 1228.684,A -85,B 0,C 180,E1 31952.835,E2 31952.835} C_VEL
LIN {X 0,Y 727.89,Z 1230.262,A -85,B 0,C 180,E1 31950.866,E2 31950.866} C_VEL
LIN {X 0,Y 727.883,Z 1230.306,A -85,B 0,C 180,E1 31949.292,E2 31949.292} C_VEL
LIN {X 0,Y 727.89,Z 1229.017,A -85,B 0,C 180,E1 31947.402,E2 31947.402} C_VEL
LIN {X 0,Y 727.917,Z 1225.972,A -85,B 0,C 180,E1 31945.509,E2 31945.509} C_VEL
LIN {X 0,Y 727.922,Z 1221.865,A -85,B 0,C 180,E1 31943.77,E2 31943.77} C_VEL
LIN {X 0,Y 727.947,Z 1215.423,A -85,B 0,C 180,E1 31941.787,E2 31941.787} C_VEL
LIN {X 0,Y 727.937,Z 1208.893,A -85,B 0,C 180,E1 31940.194,E2 31940.194} C_VEL
LIN {X 0,Y 728.023,Z 1200.298,A -85,B 0,C 180,E1 31938.433,E2 31938.433} C_VEL
LIN {X 0,Y 728.074,Z 1189.838,A -85,B 0,C 180,E1 31936.661,E2 31936.661} C_VEL
LIN {X 0,Y 728.18,Z 1179.38,A -85,B 0,C 180,E1 31935.122,E2 31935.122} C_VEL
LIN {X 0,Y 728.356,Z 1164.638,A -85,B 0,C 180,E1 31933.245,E2 31933.245} C_VEL
LIN {X 0,Y 728.507,Z 1151.299,A -85,B 0,C 180,E1 31931.764,E2 31931.764} C_VEL
LIN {X 0,Y 728.756,Z 1134.327,A -85,B 0,C 180,E1 31930.107,E2 31930.107} C_VEL
LIN {X 0,Y 729.029,Z 1117.802,A -85,B 0,C 180,E1 31928.688,E2 31928.688} C_VEL
LIN {X 0,Y 729.338,Z 1098.265,A -85,B 0,C 180,E1 31927.215,E2 31927.215} C_VEL
LIN {X 0,Y 729.683,Z 1079.776,A -85,B 0,C 180,E1 31925.986,E2 31925.986} C_VEL
LIN {X 0,Y 730.032,Z 1058.367,A -85,B 0,C 180,E1 31924.746,E2 31924.746} C_VEL
LIN {X 0,Y 730.389,Z 1038.154,A -85,B 0,C 180,E1 31923.726,E2 31923.726} C_VEL
LIN {X 0,Y 730.763,Z 1014.742,A -85,B 0,C 180,E1 31922.719,E2 31922.719} C_VEL
LIN {X 0,Y 731.033,Z 994.458,A -85,B 0,C 180,E1 31921.978,E2 31921.978} C_VEL
LIN {X 0,Y 731.402,Z 969.115,A -85,B 0,C 180,E1 31921.218,E2 31921.218} C_VEL
LIN {X 0,Y 731.603,Z 947.814,A -85,B 0,C 180,E1 31920.713,E2 31920.713} C_VEL
LIN {X 0,Y 731.872,Z 924.009,A -85,B 0,C 180,E1 31920.281,E2 31920.281} C_VEL
LIN {X 0,Y 732.026,Z 883.66,A -85,B 0,C 180,E1 31919.805,E2 31919.805} C_VEL
LIN {X 0,Y 732.717,Z 642.801,A -85,B 0,C 180,E1 31917.124,E2 31917.124} C_VEL
LIN {X 0,Y 732.929,Z 533.615,A -85,B 0,C 180,E1 31915.878,E2 31915.878} C_VEL
LIN {X 0,Y 731.737,Z 527.468,A -85,B 0,C 180,E1 31915.715,E2 31915.715} C_VEL
LIN {X 0,Y 732.112,Z 492.823,A -85,B 0,C 180,E1 31913.688,E2 31913.688} C_VEL
LIN {X 0,Y 728.206,Z 482.844,A -85,B 0,C 180,E1 31912.833,E2 31912.833} C_VEL
LIN {X 0,Y 728.125,Z 482.532,A -85,B 0,C 180,E1 31912.234,E2 31912.234} C_VEL
LIN {X 0,Y 728.096,Z 482.532,A -85,B 0,C 180,E1 31909.596,E2 31909.596} C_VEL
LIN {X 0,Y 728.153,Z 482.52,A -85,B 0,C 180,E1 31906.817,E2 31906.817} C_VEL
LIN {X 0,Y 728.115,Z 482.526,A -85,B 0,C 180,E1 31903.868,E2 31903.868} C_VEL
LIN {X 0,Y 728.103,Z 482.528,A -85,B 0,C 180,E1 31901.19,E2 31901.19} C_VEL
LIN {X 0,Y 728.156,Z 482.516,A -85,B 0,C 180,E1 31898.366,E2 31898.366} C_VEL
LIN {X 0,Y 728.108,Z 482.528,A -85,B 0,C 180,E1 31895.48,E2 31895.48} C_VEL
LIN {X 0,Y 728.113,Z 482.517,A -85,B 0,C 180,E1 31892.817,E2 31892.817} C_VEL
LIN {X 0,Y 728.158,Z 482.531,A -85,B 0,C 180,E1 31889.899,E2 31889.899} C_VEL
LIN {X 0,Y 728.106,Z 482.529,A -85,B 0,C 180,E1 31887.125,E2 31887.125} C_VEL
LIN {X 0,Y 728.13,Z 482.521,A -85,B 0,C 180,E1 31884.415,E2 31884.415} C_VEL
LIN {X 0,Y 728.139,Z 482.53,A -85,B 0,C 180,E1 31881.34,E2 31881.34} C_VEL
LIN {X 0,Y 728.108,Z 482.526,A -85,B 0,C 180,E1 31878.578,E2 31878.578} C_VEL
LIN {X 0,Y 728.155,Z 482.523,A -85,B 0,C 180,E1 31875.726,E2 31875.726} C_VEL
LIN {X 0,Y 728.118,Z 482.527,A -85,B 0,C 180,E1 31872.845,E2 31872.845} C_VEL
LIN {X 0,Y 728.129,Z 482.523,A -85,B 0,C 180,E1 31870.044,E2 31870.044} C_VEL
LIN {X 0,Y 728.147,Z 482.532,A -85,B 0,C 180,E1 31866.941,E2 31866.941} C_VEL
LIN {X 0,Y 728.112,Z 482.523,A -85,B 0,C 180,E1 31864.174,E2 31864.174} C_VEL
LIN {X 0,Y 728.155,Z 482.524,A -85,B 0,C 180,E1 31861.338,E2 31861.338} C_VEL
LIN {X 0,Y 728.123,Z 482.529,A -85,B 0,C 180,E1 31858.426,E2 31858.426} C_VEL
LIN {X 0,Y 728.136,Z 482.522,A -85,B 0,C 180,E1 31855.59,E2 31855.59} C_VEL
LIN {X 0,Y 728.148,Z 482.532,A -85,B 0,C 180,E1 31852.486,E2 31852.486} C_VEL
LIN {X 0,Y 728.121,Z 482.521,A -85,B 0,C 180,E1 31849.636,E2 31849.636} C_VEL
LIN {X 0,Y 728.15,Z 482.527,A -85,B 0,C 180,E1 31846.743,E2 31846.743} C_VEL
LIN {X 0,Y 728.153,Z 482.53,A -85,B 0,C 180,E1 31846.349,E2 31846.349} C_VEL
LIN {X 0,Y 727.143,Z 482.646,A -85,B 0,C 180,E1 31845.742,E2 31845.742} C_VEL
LIN {X 0,Y 720.702,Z 483.457,A -85,B 0,C 180,E1 31844.045,E2 31844.045} C_VEL
LIN {X 0,Y 720.179,Z 483.515,A -85,B 0,C 180,E1 31843.604,E2 31843.604} C_VEL
LIN {X 0,Y 720.213,Z 483.509,A -85,B 0,C 180,E1 31840.739,E2 31840.739} C_VEL
LIN {X 0,Y 720.191,Z 483.515,A -85,B 0,C 180,E1 31837.813,E2 31837.813} C_VEL
LIN {X 0,Y 720.216,Z 483.51,A -85,B 0,C 180,E1 31834.844,E2 31834.844} C_VEL
LIN {X 0,Y 720.202,Z 483.521,A -85,B 0,C 180,E1 31831.743,E2 31831.743} C_VEL
LIN {X 0,Y 720.207,Z 483.51,A -85,B 0,C 180,E1 31828.78,E2 31828.78} C_VEL
LIN {X 0,Y 720.213,Z 483.521,A -85,B 0,C 180,E1 31825.69,E2 31825.69} C_VEL
LIN {X 0,Y 720.194,Z 483.503,A -85,B 0,C 180,E1 31822.747,E2 31822.747} C_VEL
LIN {X 0,Y 720.211,Z 483.518,A -85,B 0,C 180,E1 31819.779,E2 31819.779} C_VEL
LIN {X 0,Y 720.186,Z 483.51,A -85,B 0,C 180,E1 31816.908,E2 31816.908} C_VEL
LIN {X 0,Y 720.211,Z 483.513,A -85,B 0,C 180,E1 31814.015,E2 31814.015} C_VEL
LIN {X 0,Y 720.201,Z 483.521,A -85,B 0,C 180,E1 31811.046,E2 31811.046} C_VEL
LIN {X 0,Y 720.218,Z 483.518,A -85,B 0,C 180,E1 31808.053,E2 31808.053} C_VEL
LIN {X 0,Y 720.256,Z 483.77,A -85,B 0,C 180,E1 31807.206,E2 31807.206} C_VEL
LIN {X 0,Y 724.977,Z 496.375,A -85,B 0,C 180,E1 31806.078,E2 31806.078} C_VEL
LIN {X 0,Y 724.235,Z 541.07,A -85,B 0,C 180,E1 31803.283,E2 31803.283} C_VEL
LIN {X 0,Y 723.551,Z 587.361,A -85,B 0,C 180,E1 31800.474,E2 31800.474} C_VEL
LIN {X 0,Y 722.932,Z 633.873,A -85,B 0,C 180,E1 31797.725,E2 31797.725} C_VEL
LIN {X 0,Y 722.787,Z 651.297,A -85,B 0,C 180,E1 31796.717,E2 31796.717} C_VEL
LIN {X 0,Y 723.867,Z 659.143,A -85,B 0,C 180,E1 31796.577,E2 31796.577} C_VEL
LIN {X 0,Y 723.072,Z 934.26,A -85,B 0,C 180,E1 31793.651,E2 31793.651} C_VEL
LIN {X 0,Y 722.905,Z 962.513,A -85,B 0,C 180,E1 31793.301,E2 31793.301} C_VEL
LIN {X 0,Y 722.746,Z 984.088,A -85,B 0,C 180,E1 31792.891,E2 31792.891} C_VEL
LIN {X 0,Y 722.478,Z 1004.837,A -85,B 0,C 180,E1 31792.348,E2 31792.348} C_VEL
LIN {X 0,Y 722.19,Z 1025.856,A -85,B 0,C 180,E1 31791.652,E2 31791.652} C_VEL
LIN {X 0,Y 721.918,Z 1045.632,A -85,B 0,C 180,E1 31790.851,E2 31790.851} C_VEL
LIN {X 0,Y 721.571,Z 1065.208,A -85,B 0,C 180,E1 31789.893,E2 31789.893} C_VEL
LIN {X 0,Y 721.246,Z 1084.069,A -85,B 0,C 180,E1 31788.803,E2 31788.803} C_VEL
LIN {X 0,Y 720.96,Z 1101.878,A -85,B 0,C 180,E1 31787.598,E2 31787.598} C_VEL
LIN {X 0,Y 720.7,Z 1118.661,A -85,B 0,C 180,E1 31786.275,E2 31786.275} C_VEL
LIN {X 0,Y 720.466,Z 1133.793,A -85,B 0,C 180,E1 31784.877,E2 31784.877} C_VEL
LIN {X 0,Y 720.268,Z 1147.477,A -85,B 0,C 180,E1 31783.405,E2 31783.405} C_VEL
LIN {X 0,Y 720.134,Z 1159.765,A -85,B 0,C 180,E1 31781.858,E2 31781.858} C_VEL
LIN {X 0,Y 720.045,Z 1170.105,A -85,B 0,C 180,E1 31780.319,E2 31780.319} C_VEL
LIN {X 0,Y 719.979,Z 1179.06,A -85,B 0,C 180,E1 31778.706,E2 31778.706} C_VEL
LIN {X 0,Y 719.939,Z 1186.686,A -85,B 0,C 180,E1 31777.02,E2 31777.02} C_VEL
LIN {X 0,Y 719.923,Z 1192.524,A -85,B 0,C 180,E1 31775.339,E2 31775.339} C_VEL
LIN {X 0,Y 719.914,Z 1196.695,A -85,B 0,C 180,E1 31773.663,E2 31773.663} C_VEL
LIN {X 0,Y 719.917,Z 1199.441,A -85,B 0,C 180,E1 31771.91,E2 31771.91} C_VEL
LIN {X 0,Y 719.907,Z 1200.448,A -85,B 0,C 180,E1 31770.159,E2 31770.159} C_VEL
LIN {X 0,Y 719.903,Z 1199.787,A -85,B 0,C 180,E1 31768.408,E2 31768.408} C_VEL
LIN {X 0,Y 719.904,Z 1197.503,A -85,B 0,C 180,E1 31766.656,E2 31766.656} C_VEL
LIN {X 0,Y 719.913,Z 1193.695,A -85,B 0,C 180,E1 31764.98,E2 31764.98} C_VEL
LIN {X 0,Y 719.92,Z 1188.237,A -85,B 0,C 180,E1 31763.3,E2 31763.3} C_VEL
LIN {X 0,Y 719.977,Z 1181.137,A -85,B 0,C 180,E1 31761.615,E2 31761.615} C_VEL
LIN {X 0,Y 720.023,Z 1172.55,A -85,B 0,C 180,E1 31760.004,E2 31760.004} C_VEL
LIN {X 0,Y 720.108,Z 1162.137,A -85,B 0,C 180,E1 31758.385,E2 31758.385} C_VEL
LIN {X 0,Y 720.249,Z 1150.358,A -85,B 0,C 180,E1 31756.84,E2 31756.84} C_VEL
LIN {X 0,Y 720.429,Z 1136.693,A -85,B 0,C 180,E1 31755.325,E2 31755.325} C_VEL
LIN {X 0,Y 720.615,Z 1122.45,A -85,B 0,C 180,E1 31753.972,E2 31753.972} C_VEL
LIN {X 0,Y 720.878,Z 1105.863,A -85,B 0,C 180,E1 31752.61,E2 31752.61} C_VEL
LIN {X 0,Y 721.188,Z 1088.448,A -85,B 0,C 180,E1 31751.383,E2 31751.383} C_VEL
LIN {X 0,Y 721.502,Z 1070.052,A -85,B 0,C 180,E1 31750.279,E2 31750.279} C_VEL
LIN {X 0,Y 721.795,Z 1051.14,A -85,B 0,C 180,E1 31749.315,E2 31749.315} C_VEL
LIN {X 0,Y 722.132,Z 1030.838,A -85,B 0,C 180,E1 31748.446,E2 31748.446} C_VEL
LIN {X 0,Y 722.413,Z 1010.755,A -85,B 0,C 180,E1 31747.74,E2 31747.74} C_VEL
LIN {X 0,Y 722.663,Z 989.451,A -85,B 0,C 180,E1 31747.149,E2 31747.149} C_VEL
LIN {X 0,Y 722.886,Z 967.255,A -85,B 0,C 180,E1 31746.687,E2 31746.687} C_VEL
LIN {X 0,Y 723.028,Z 945.741,A -85,B 0,C 180,E1 31746.382,E2 31746.382} C_VEL
LIN {X 0,Y 723.827,Z 672.389,A -85,B 0,C 180,E1 31743.475,E2 31743.475} C_VEL
LIN {X 0,Y 723.646,Z 656.345,A -85,B 0,C 180,E1 31743.294,E2 31743.294} C_VEL
LIN {X 0,Y 722.79,Z 651.335,A -85,B 0,C 180,E1 31743.194,E2 31743.194} C_VEL
LIN {X 0,Y 723.353,Z 602.53,A -85,B 0,C 180,E1 31740.34,E2 31740.34} C_VEL
LIN {X 0,Y 723.993,Z 556.106,A -85,B 0,C 180,E1 31737.548,E2 31737.548} C_VEL
LIN {X 0,Y 724.79,Z 507.625,A -85,B 0,C 180,E1 31734.544,E2 31734.544} C_VEL
LIN {X 0,Y 724.902,Z 495.886,A -85,B 0,C 180,E1 31733.796,E2 31733.796} C_VEL
LIN {X 0,Y 720.248,Z 483.751,A -85,B 0,C 180,E1 31732.7,E2 31732.7} C_VEL
LIN {X 0,Y 720.199,Z 483.512,A -85,B 0,C 180,E1 31729.659,E2 31729.659} C_VEL
LIN {X 0,Y 720.204,Z 483.509,A -85,B 0,C 180,E1 31726.7,E2 31726.7} C_VEL
LIN {X 0,Y 720.205,Z 483.506,A -85,B 0,C 180,E1 31723.557,E2 31723.557} C_VEL
LIN {X 0,Y 720.198,Z 483.519,A -85,B 0,C 180,E1 31720.588,E2 31720.588} C_VEL
LIN {X 0,Y 720.216,Z 483.502,A -85,B 0,C 180,E1 31717.552,E2 31717.552} C_VEL
LIN {X 0,Y 720.18,Z 483.518,A -85,B 0,C 180,E1 31714.697,E2 31714.697} C_VEL
LIN {X 0,Y 720.213,Z 483.517,A -85,B 0,C 180,E1 31711.829,E2 31711.829} C_VEL
LIN {X 0,Y 720.188,Z 483.513,A -85,B 0,C 180,E1 31708.983,E2 31708.983} C_VEL
LIN {X 0,Y 720.206,Z 483.518,A -85,B 0,C 180,E1 31706.074,E2 31706.074} C_VEL
LIN {X 0,Y 720.201,Z 483.507,A -85,B 0,C 180,E1 31702.962,E2 31702.962} C_VEL
LIN {X 0,Y 720.183,Z 483.519,A -85,B 0,C 180,E1 31700.14,E2 31700.14} C_VEL
LIN {X 0,Y 720.215,Z 483.514,A -85,B 0,C 180,E1 31697.2,E2 31697.2} C_VEL
LIN {X 0,Y 720.175,Z 483.511,A -85,B 0,C 180,E1 31694.39,E2 31694.39} C_VEL
LIN {X 0,Y 720.213,Z 483.521,A -85,B 0,C 180,E1 31691.532,E2 31691.532} C_VEL
LIN {X 0,Y 720.191,Z 483.512,A -85,B 0,C 180,E1 31688.463,E2 31688.463} C_VEL
LIN {X 0,Y 720.182,Z 483.516,A -85,B 0,C 180,E1 31685.657,E2 31685.657} C_VEL
LIN {X 0,Y 720.218,Z 483.511,A -85,B 0,C 180,E1 31682.706,E2 31682.706} C_VEL
LIN {X 0,Y 720.171,Z 483.514,A -85,B 0,C 180,E1 31679.92,E2 31679.92} C_VEL
LIN {X 0,Y 720.208,Z 483.52,A -85,B 0,C 180,E1 31677.135,E2 31677.135} C_VEL
LIN {X 0,Y 720.193,Z 483.512,A -85,B 0,C 180,E1 31674.103,E2 31674.103} C_VEL
LIN {X 0,Y 720.171,Z 483.513,A -85,B 0,C 180,E1 31671.376,E2 31671.376} C_VEL
LIN {X 0,Y 720.217,Z 483.514,A -85,B 0,C 180,E1 31668.549,E2 31668.549} C_VEL
LIN {X 0,Y 720.175,Z 483.514,A -85,B 0,C 180,E1 31665.692,E2 31665.692} C_VEL
LIN {X 0,Y 720.177,Z 483.517,A -85,B 0,C 180,E1 31662.965,E2 31662.965} C_VEL
LIN {X 0,Y 720.217,Z 483.509,A -85,B 0,C 180,E1 31659.945,E2 31659.945} C_VEL
LIN {X 0,Y 720.163,Z 483.517,A -85,B 0,C 180,E1 31657.123,E2 31657.123} C_VEL
LIN {X 0,Y 720.218,Z 483.52,A -85,B 0,C 180,E1 31654.288,E2 31654.288} C_VEL
LIN {X 0,Y 720.172,Z 483.513,A -85,B 0,C 180,E1 31651.289,E2 31651.289} C_VEL
LIN {X 0,Y 720.17,Z 483.519,A -85,B 0,C 180,E1 31648.624,E2 31648.624} C_VEL
LIN {X 0,Y 720.217,Z 483.513,A -85,B 0,C 180,E1 31645.691,E2 31645.691} C_VEL
LIN {X 0,Y 720.162,Z 483.517,A -85,B 0,C 180,E1 31642.845,E2 31642.845} C_VEL
LIN {X 0,Y 720.186,Z 483.509,A -85,B 0,C 180,E1 31640.152,E2 31640.152} C_VEL
LIN {X 0,Y 720.183,Z 483.508,A -85,B 0,C 180,E1 31637.023,E2 31637.023} C_VEL
LIN {X 0,Y 720.16,Z 483.52,A -85,B 0,C 180,E1 31634.353,E2 31634.353} C_VEL
LIN {X 0,Y 720.22,Z 483.508,A -85,B 0,C 180,E1 31631.556,E2 31631.556} C_VEL
LIN {X 0,Y 720.165,Z 483.52,A -85,B 0,C 180,E1 31628.585,E2 31628.585} C_VEL
LIN {X 0,Y 720.249,Z 483.798,A -85,B 0,C 180,E1 31627.593,E2 31627.593} C_VEL
LIN {X 0,Y 725.235,Z 497.044,A -85,B 0,C 180,E1 31626.456,E2 31626.456} C_VEL
LIN {X 0,Y 724.781,Z 527.984,A -85,B 0,C 180,E1 31624.636,E2 31624.636} C_VEL
LIN {X 0,Y 726.477,Z 537.117,A -85,B 0,C 180,E1 31624.427,E2 31624.427} C_VEL
LIN {X 0,Y 725.418,Z 794.213,A -85,B 0,C 180,E1 31621.511,E2 31621.511} C_VEL
LIN {X 0,Y 724.937,Z 919.046,A -85,B 0,C 180,E1 31620.099,E2 31620.099} C_VEL
LIN {X 0,Y 724.612,Z 944.69,A -85,B 0,C 180,E1 31619.665,E2 31619.665} C_VEL
LIN {X 0,Y 724.342,Z 966.272,A -85,B 0,C 180,E1 31619.164,E2 31619.164} C_VEL
LIN {X 0,Y 724.022,Z 989.317,A -85,B 0,C 180,E1 31618.498,E2 31618.498} C_VEL
LIN {X 0,Y 723.548,Z 1012.508,A -85,B 0,C 180,E1 31617.666,E2 31617.666} C_VEL
LIN {X 0,Y 723.146,Z 1035.199,A -85,B 0,C 180,E1 31616.703,E2 31616.703} C_VEL
LIN {X 0,Y 722.634,Z 1056.769,A -85,B 0,C 180,E1 31615.619,E2 31615.619} C_VEL
LIN {X 0,Y 722.216,Z 1077.849,A -85,B 0,C 180,E1 31614.404,E2 31614.404} C_VEL
LIN {X 0,Y 721.742,Z 1097.576,A -85,B 0,C 180,E1 31613.088,E2 31613.088} C_VEL
LIN {X 0,Y 721.363,Z 1116.787,A -85,B 0,C 180,E1 31611.635,E2 31611.635} C_VEL
LIN {X 0,Y 721.007,Z 1133.399,A -85,B 0,C 180,E1 31610.2,E2 31610.2} C_VEL
LIN {X 0,Y 720.711,Z 1150.524,A -85,B 0,C 180,E1 31608.524,E2 31608.524} C_VEL
LIN {X 0,Y 720.475,Z 1164.009,A -85,B 0,C 180,E1 31607.018,E2 31607.018} C_VEL
LIN {X 0,Y 720.273,Z 1178.222,A -85,B 0,C 180,E1 31605.21,E2 31605.21} C_VEL
LIN {X 0,Y 720.137,Z 1189.318,A -85,B 0,C 180,E1 31603.571,E2 31603.571} C_VEL
LIN {X 0,Y 720.047,Z 1199.956,A -85,B 0,C 180,E1 31601.762,E2 31601.762} C_VEL
LIN {X 0,Y 719.952,Z 1208.894,A -85,B 0,C 180,E1 31599.916,E2 31599.916} C_VEL
LIN {X 0,Y 719.953,Z 1215.424,A -85,B 0,C 180,E1 31598.304,E2 31598.304} C_VEL
LIN {X 0,Y 719.924,Z 1222.071,A -85,B 0,C 180,E1 31596.219,E2 31596.219} C_VEL
LIN {X 0,Y 719.917,Z 1226.131,A -85,B 0,C 180,E1 31594.461,E2 31594.461} C_VEL
LIN {X 0,Y 719.894,Z 1229.093,A -85,B 0,C 180,E1 31592.547,E2 31592.547} C_VEL
LIN {X 0,Y 719.883,Z 1230.306,A -85,B 0,C 180,E1 31590.716,E2 31590.716} C_VEL
LIN {X 0,Y 719.896,Z 1230.24,A -85,B 0,C 180,E1 31589.045,E2 31589.045} C_VEL
LIN {X 0,Y 719.882,Z 1228.559,A -85,B 0,C 180,E1 31587.045,E2 31587.045} C_VEL
LIN {X 0,Y 719.916,Z 1225.813,A -85,B 0,C 180,E1 31585.38,E2 31585.38} C_VEL
LIN {X 0,Y 719.92,Z 1221.245,A -85,B 0,C 180,E1 31583.461,E2 31583.461} C_VEL
LIN {X 0,Y 719.942,Z 1214.816,A -85,B 0,C 180,E1 31581.535,E2 31581.535} C_VEL
LIN {X 0,Y 719.962,Z 1208.183,A -85,B 0,C 180,E1 31579.922,E2 31579.922} C_VEL
LIN {X 0,Y 720.046,Z 1198.494,A -85,B 0,C 180,E1 31577.978,E2 31577.978} C_VEL
LIN {X 0,Y 720.146,Z 1188.8,A -85,B 0,C 180,E1 31576.348,E2 31576.348} C_VEL
LIN {X 0,Y 720.304,Z 1176.447,A -85,B 0,C 180,E1 31574.543,E2 31574.543} C_VEL
LIN {X 0,Y 720.482,Z 1163.225,A -85,B 0,C 180,E1 31572.89,E2 31572.89} C_VEL
LIN {X 0,Y 720.774,Z 1148.183,A -85,B 0,C 180,E1 31571.226,E2 31571.226} C_VEL
LIN {X 0,Y 721.053,Z 1131.541,A -85,B 0,C 180,E1 31569.632,E2 31569.632} C_VEL
LIN {X 0,Y 721.426,Z 1113.615,A -85,B 0,C 180,E1 31568.11,E2 31568.11} C_VEL
LIN {X 0,Y 721.81,Z 1095.249,A -85,B 0,C 180,E1 31566.748,E2 31566.748} C_VEL
LIN {X 0,Y 722.275,Z 1073.451,A -85,B 0,C 180,E1 31565.331,E2 31565.331} C_VEL
LIN {X 0,Y 722.731,Z 1053.545,A -85,B 0,C 180,E1 31564.209,E2 31564.209} C_VEL
LIN {X 0,Y 723.207,Z 1030.279,A -85,B 0,C 180,E1 31563.078,E2 31563.078} C_VEL
LIN {X 0,Y 723.627,Z 1009.136,A -85,B 0,C 180,E1 31562.203,E2 31562.203} C_VEL
LIN {X 0,Y 724.074,Z 984.999,A -85,B 0,C 180,E1 31561.369,E2 31561.369} C_VEL
LIN {X 0,Y 724.363,Z 963.145,A -85,B 0,C 180,E1 31560.755,E2 31560.755} C_VEL
LIN {X 0,Y 724.745,Z 938.512,A -85,B 0,C 180,E1 31560.213,E2 31560.213} C_VEL
LIN {X 0,Y 724.95,Z 915.774,A -85,B 0,C 180,E1 31559.858,E2 31559.858} C_VEL
LIN {X 0,Y 725.929,Z 658.578,A -85,B 0,C 180,E1 31556.959,E2 31556.959} C_VEL
LIN {X 0,Y 726.282,Z 535.197,A -85,B 0,C 180,E1 31555.54,E2 31555.54} C_VEL
LIN {X 0,Y 724.765,Z 527.485,A -85,B 0,C 180,E1 31555.339,E2 31555.339} C_VEL
LIN {X 0,Y 725.181,Z 496.364,A -85,B 0,C 180,E1 31553.5,E2 31553.5} C_VEL
LIN {X 0,Y 720.244,Z 483.773,A -85,B 0,C 180,E1 31552.402,E2 31552.402} C_VEL
LIN {X 0,Y 720.16,Z 483.524,A -85,B 0,C 180,E1 31549.786,E2 31549.786} C_VEL
LIN {X 0,Y 720.179,Z 483.509,A -85,B 0,C 180,E1 31547.134,E2 31547.134} C_VEL
LIN {X 0,Y 720.191,Z 483.51,A -85,B 0,C 180,E1 31544.016,E2 31544.016} C_VEL
LIN {X 0,Y 720.162,Z 483.518,A -85,B 0,C 180,E1 31541.262,E2 31541.262} C_VEL
LIN {X 0,Y 720.22,Z 483.501,A -85,B 0,C 180,E1 31538.46,E2 31538.46} C_VEL
LIN {X 0,Y 720.174,Z 483.518,A -85,B 0,C 180,E1 31535.553,E2 31535.553} C_VEL
LIN {X 0,Y 720.171,Z 483.504,A -85,B 0,C 180,E1 31532.865,E2 31532.865} C_VEL
LIN {X 0,Y 720.22,Z 483.52,A -85,B 0,C 180,E1 31529.895,E2 31529.895} C_VEL
LIN {X 0,Y 720.166,Z 483.518,A -85,B 0,C 180,E1 31527.091,E2 31527.091} C_VEL
LIN {X 0,Y 720.199,Z 483.509,A -85,B 0,C 180,E1 31524.352,E2 31524.352} C_VEL
LIN {X 0,Y 720.19,Z 483.518,A -85,B 0,C 180,E1 31521.246,E2 31521.246} C_VEL
LIN {X 0,Y 720.175,Z 483.514,A -85,B 0,C 180,E1 31518.455,E2 31518.455} C_VEL
LIN {X 0,Y 720.216,Z 483.515,A -85,B 0,C 180,E1 31515.537,E2 31515.537} C_VEL
LIN {X 0,Y 720.171,Z 483.514,A -85,B 0,C 180,E1 31512.672,E2 31512.672} C_VEL
LIN {X 0,Y 720.214,Z 483.511,A -85,B 0,C 180,E1 31509.832,E2 31509.832} C_VEL
LIN {X 0,Y 720.19,Z 483.52,A -85,B 0,C 180,E1 31506.777,E2 31506.777} C_VEL
LIN {X 0,Y 720.181,Z 483.51,A -85,B 0,C 180,E1 31503.981,E2 31503.981} C_VEL
LIN {X 0,Y 720.218,Z 483.518,A -85,B 0,C 180,E1 31501.034,E2 31501.034} C_VEL
LIN {X 0,Y 720.173,Z 483.515,A -85,B 0,C 180,E1 31498.17,E2 31498.17} C_VEL
LIN {X 0,Y 720.219,Z 483.51,A -85,B 0,C 180,E1 31495.302,E2 31495.302} C_VEL
LIN {X 0,Y 720.188,Z 483.519,A -85,B 0,C 180,E1 31492.26,E2 31492.26} C_VEL
LIN {X 0,Y 720.204,Z 483.506,A -85,B 0,C 180,E1 31489.359,E2 31489.359} C_VEL
LIN {X 0,Y 720.207,Z 483.517,A -85,B 0,C 180,E1 31486.266,E2 31486.266} C_VEL
LIN {X 0,Y 720.179,Z 483.515,A -85,B 0,C 180,E1 31483.604,E2 31483.604} C_VEL
LIN {X 0,Y 719.211,Z 483.638,A -85,B 0,C 180,E1 31482.991,E2 31482.991} C_VEL
LIN {X 0,Y 712.822,Z 484.429,A -85,B 0,C 180,E1 31481.274,E2 31481.274} C_VEL
LIN {X 0,Y 712.276,Z 484.497,A -85,B 0,C 180,E1 31480.828,E2 31480.828} C_VEL
LIN {X 0,Y 712.252,Z 484.504,A -85,B 0,C 180,E1 31477.813,E2 31477.813} C_VEL
LIN {X 0,Y 712.273,Z 484.5,A -85,B 0,C 180,E1 31474.88,E2 31474.88} C_VEL
LIN {X 0,Y 712.265,Z 484.51,A -85,B 0,C 180,E1 31471.765,E2 31471.765} C_VEL
LIN {X 0,Y 712.266,Z 484.5,A -85,B 0,C 180,E1 31468.801,E2 31468.801} C_VEL
LIN {X 0,Y 712.271,Z 484.511,A -85,B 0,C 180,E1 31465.644,E2 31465.644} C_VEL
LIN {X 0,Y 712.262,Z 484.49,A -85,B 0,C 180,E1 31462.666,E2 31462.666} C_VEL
LIN {X 0,Y 712.278,Z 484.511,A -85,B 0,C 180,E1 31459.567,E2 31459.567} C_VEL
LIN {X 0,Y 712.253,Z 484.496,A -85,B 0,C 180,E1 31456.648,E2 31456.648} C_VEL
LIN {X 0,Y 712.269,Z 484.503,A -85,B 0,C 180,E1 31453.7,E2 31453.7} C_VEL
LIN {X 0,Y 712.25,Z 484.508,A -85,B 0,C 180,E1 31450.828,E2 31450.828} C_VEL
LIN {X 0,Y 712.278,Z 484.507,A -85,B 0,C 180,E1 31447.914,E2 31447.914} C_VEL
LIN {X 0,Y 712.339,Z 484.981,A -85,B 0,C 180,E1 31447.6,E2 31447.6} C_VEL
LIN {X 0,Y 718.01,Z 499.809,A -85,B 0,C 180,E1 31446.263,E2 31446.263} C_VEL
LIN {X 0,Y 717.119,Z 544.914,A -85,B 0,C 180,E1 31443.417,E2 31443.417} C_VEL
LIN {X 0,Y 716.274,Z 591.168,A -85,B 0,C 180,E1 31440.585,E2 31440.585} C_VEL
LIN {X 0,Y 715.55,Z 636.73,A -85,B 0,C 180,E1 31437.866,E2 31437.866} C_VEL
LIN {X 0,Y 715.411,Z 651.338,A -85,B 0,C 180,E1 31437.015,E2 31437.015} C_VEL
LIN {X 0,Y 716.708,Z 660.339,A -85,B 0,C 180,E1 31436.851,E2 31436.851} C_VEL
LIN {X 0,Y 715.74,Z 935.202,A -85,B 0,C 180,E1 31433.898,E2 31433.898} C_VEL
LIN {X 0,Y 715.543,Z 962.939,A -85,B 0,C 180,E1 31433.549,E2 31433.549} C_VEL
LIN {X 0,Y 715.344,Z 984.467,A -85,B 0,C 180,E1 31433.132,E2 31433.132} C_VEL
LIN {X 0,Y 715.024,Z 1005.593,A -85,B 0,C 180,E1 31432.572,E2 31432.572} C_VEL
LIN {X 0,Y 714.663,Z 1026.997,A -85,B 0,C 180,E1 31431.848,E2 31431.848} C_VEL
LIN {X 0,Y 714.305,Z 1047.441,A -85,B 0,C 180,E1 31430.998,E2 31430.998} C_VEL
LIN {X 0,Y 713.912,Z 1066.921,A -85,B 0,C 180,E1 31430.025,E2 31430.025} C_VEL
LIN {X 0,Y 713.516,Z 1085.407,A -85,B 0,C 180,E1 31428.929,E2 31428.929} C_VEL
LIN {X 0,Y 713.156,Z 1103.548,A -85,B 0,C 180,E1 31427.67,E2 31427.67} C_VEL
LIN {X 0,Y 712.853,Z 1119.595,A -85,B 0,C 180,E1 31426.375,E2 31426.375} C_VEL
LIN {X 0,Y 712.579,Z 1134.642,A -85,B 0,C 180,E1 31424.962,E2 31424.962} C_VEL
LIN {X 0,Y 712.344,Z 1148.186,A -85,B 0,C 180,E1 31423.474,E2 31423.474} C_VEL
LIN {X 0,Y 712.17,Z 1160.924,A -85,B 0,C 180,E1 31421.828,E2 31421.828} C_VEL
LIN {X 0,Y 712.067,Z 1171.119,A -85,B 0,C 180,E1 31420.272,E2 31420.272} C_VEL
LIN {X 0,Y 711.99,Z 1179.928,A -85,B 0,C 180,E1 31418.631,E2 31418.631} C_VEL
LIN {X 0,Y 711.931,Z 1187.597,A -85,B 0,C 180,E1 31416.856,E2 31416.856} C_VEL
LIN {X 0,Y 711.926,Z 1193.256,A -85,B 0,C 180,E1 31415.157,E2 31415.157} C_VEL
LIN {X 0,Y 711.912,Z 1197.169,A -85,B 0,C 180,E1 31413.462,E2 31413.462} C_VEL
LIN {X 0,Y 711.908,Z 1199.711,A -85,B 0,C 180,E1 31411.61,E2 31411.61} C_VEL
LIN {X 0,Y 711.914,Z 1200.495,A -85,B 0,C 180,E1 31409.92,E2 31409.92} C_VEL
LIN {X 0,Y 711.917,Z 1199.586,A -85,B 0,C 180,E1 31408.149,E2 31408.149} C_VEL
LIN {X 0,Y 711.916,Z 1197.029,A -85,B 0,C 180,E1 31406.376,E2 31406.376} C_VEL
LIN {X 0,Y 711.923,Z 1193.059,A -85,B 0,C 180,E1 31404.681,E2 31404.681} C_VEL
LIN {X 0,Y 711.936,Z 1187.328,A -85,B 0,C 180,E1 31402.982,E2 31402.982} C_VEL
LIN {X 0,Y 711.99,Z 1179.512,A -85,B 0,C 180,E1 31401.195,E2 31401.195} C_VEL
LIN {X 0,Y 712.078,Z 1170.675,A -85,B 0,C 180,E1 31399.564,E2 31399.564} C_VEL
LIN {X 0,Y 712.177,Z 1160.403,A -85,B 0,C 180,E1 31398.008,E2 31398.008} C_VEL
LIN {X 0,Y 712.345,Z 1148.248,A -85,B 0,C 180,E1 31396.444,E2 31396.444} C_VEL
LIN {X 0,Y 712.578,Z 1134.712,A -85,B 0,C 180,E1 31394.955,E2 31394.955} C_VEL
LIN {X 0,Y 712.848,Z 1119.661,A -85,B 0,C 180,E1 31393.541,E2 31393.541} C_VEL
LIN {X 0,Y 713.156,Z 1103.627,A -85,B 0,C 180,E1 31392.246,E2 31392.246} C_VEL
LIN {X 0,Y 713.516,Z 1085.486,A -85,B 0,C 180,E1 31390.986,E2 31390.986} C_VEL
LIN {X 0,Y 713.91,Z 1067.011,A -85,B 0,C 180,E1 31389.89,E2 31389.89} C_VEL
LIN {X 0,Y 714.304,Z 1047.525,A -85,B 0,C 180,E1 31388.916,E2 31388.916} C_VEL
LIN {X 0,Y 714.661,Z 1027.099,A -85,B 0,C 180,E1 31388.065,E2 31388.065} C_VEL
LIN {X 0,Y 715.023,Z 1005.851,A -85,B 0,C 180,E1 31387.345,E2 31387.345} C_VEL
LIN {X 0,Y 715.342,Z 984.496,A -85,B 0,C 180,E1 31386.778,E2 31386.778} C_VEL
LIN {X 0,Y 715.544,Z 963.035,A -85,B 0,C 180,E1 31386.363,E2 31386.363} C_VEL
LIN {X 0,Y 715.742,Z 935.387,A -85,B 0,C 180,E1 31386.014,E2 31386.014} C_VEL
LIN {X 0,Y 716.706,Z 658.803,A -85,B 0,C 180,E1 31383.042,E2 31383.042} C_VEL
LIN {X 0,Y 715.409,Z 651.34,A -85,B 0,C 180,E1 31382.895,E2 31382.895} C_VEL
LIN {X 0,Y 716.083,Z 603.28,A -85,B 0,C 180,E1 31380.055,E2 31380.055} C_VEL
LIN {X 0,Y 716.879,Z 556.964,A -85,B 0,C 180,E1 31377.238,E2 31377.238} C_VEL
LIN {X 0,Y 717.821,Z 509.168,A -85,B 0,C 180,E1 31374.245,E2 31374.245} C_VEL
LIN {X 0,Y 717.94,Z 499.303,A -85,B 0,C 180,E1 31373.61,E2 31373.61} C_VEL
LIN {X 0,Y 712.319,Z 484.837,A -85,B 0,C 180,E1 31372.291,E2 31372.291} C_VEL
LIN {X 0,Y 712.245,Z 484.498,A -85,B 0,C 180,E1 31371.44,E2 31371.44} C_VEL
LIN {X 0,Y 712.28,Z 484.506,A -85,B 0,C 180,E1 31368.558,E2 31368.558} C_VEL
LIN {X 0,Y 712.256,Z 484.503,A -85,B 0,C 180,E1 31365.492,E2 31365.492} C_VEL
LIN {X 0,Y 712.265,Z 484.496,A -85,B 0,C 180,E1 31362.582,E2 31362.582} C_VEL
LIN {X 0,Y 712.268,Z 484.498,A -85,B 0,C 180,E1 31359.46,E2 31359.46} C_VEL
LIN {X 0,Y 712.253,Z 484.499,A -85,B 0,C 180,E1 31356.529,E2 31356.529} C_VEL
LIN {X 0,Y 712.279,Z 484.497,A -85,B 0,C 180,E1 31353.483,E2 31353.483} C_VEL
LIN {X 0,Y 712.24,Z 484.506,A -85,B 0,C 180,E1 31350.623,E2 31350.623} C_VEL
LIN {X 0,Y 712.276,Z 484.505,A -85,B 0,C 180,E1 31347.779,E2 31347.779} C_VEL
LIN {X 0,Y 712.245,Z 484.503,A -85,B 0,C 180,E1 31344.819,E2 31344.819} C_VEL
LIN {X 0,Y 712.266,Z 484.506,A -85,B 0,C 180,E1 31341.927,E2 31341.927} C_VEL
LIN {X 0,Y 712.261,Z 484.496,A -85,B 0,C 180,E1 31338.837,E2 31338.837} C_VEL
LIN {X 0,Y 712.246,Z 484.508,A -85,B 0,C 180,E1 31335.971,E2 31335.971} C_VEL
LIN {X 0,Y 712.279,Z 484.501,A -85,B 0,C 180,E1 31332.98,E2 31332.98} C_VEL
LIN {X 0,Y 712.233,Z 484.5,A -85,B 0,C 180,E1 31330.107,E2 31330.107} C_VEL
LIN {X 0,Y 712.281,Z 484.506,A -85,B 0,C 180,E1 31327.258,E2 31327.258} C_VEL
LIN {X 0,Y 712.245,Z 484.502,A -85,B 0,C 180,E1 31324.267,E2 31324.267} C_VEL
LIN {X 0,Y 712.249,Z 484.508,A -85,B 0,C 180,E1 31321.448,E2 31321.448} C_VEL
LIN {X 0,Y 712.273,Z 484.5,A -85,B 0,C 180,E1 31318.391,E2 31318.391} C_VEL
LIN {X 0,Y 712.231,Z 484.503,A -85,B 0,C 180,E1 31315.572,E2 31315.572} C_VEL
LIN {X 0,Y 712.279,Z 484.502,A -85,B 0,C 180,E1 31312.742,E2 31312.742} C_VEL
LIN {X 0,Y 712.237,Z 484.504,A -85,B 0,C 180,E1 31309.763,E2 31309.763} C_VEL
LIN {X 0,Y 712.255,Z 484.505,A -85,B 0,C 180,E1 31306.937,E2 31306.937} C_VEL
LIN {X 0,Y 712.249,Z 484.499,A -85,B 0,C 180,E1 31303.781,E2 31303.781} C_VEL
LIN {X 0,Y 712.235,Z 484.508,A -85,B 0,C 180,E1 31300.992,E2 31300.992} C_VEL
LIN {X 0,Y 712.284,Z 484.502,A -85,B 0,C 180,E1 31297.987,E2 31297.987} C_VEL
LIN {X 0,Y 712.226,Z 484.501,A -85,B 0,C 180,E1 31295.18,E2 31295.18} C_VEL
LIN {X 0,Y 712.27,Z 484.51,A -85,B 0,C 180,E1 31292.347,E2 31292.347} C_VEL
LIN {X 0,Y 712.238,Z 484.503,A -85,B 0,C 180,E1 31289.269,E2 31289.269} C_VEL
LIN {X 0,Y 712.233,Z 484.495,A -85,B 0,C 180,E1 31286.514,E2 31286.514} C_VEL
LIN {X 0,Y 712.275,Z 484.502,A -85,B 0,C 180,E1 31283.472,E2 31283.472} C_VEL
LIN {X 0,Y 712.219,Z 484.492,A -85,B 0,C 180,E1 31280.672,E2 31280.672} C_VEL
LIN {X 0,Y 712.276,Z 484.507,A -85,B 0,C 180,E1 31277.854,E2 31277.854} C_VEL
LIN {X 0,Y 712.234,Z 484.506,A -85,B 0,C 180,E1 31274.849,E2 31274.849} C_VEL
LIN {X 0,Y 712.225,Z 484.498,A -85,B 0,C 180,E1 31272.147,E2 31272.147} C_VEL
LIN {X 0,Y 712.281,Z 484.496,A -85,B 0,C 180,E1 31269.205,E2 31269.205} C_VEL
LIN {X 0,Y 712.253,Z 484.721,A -85,B 0,C 180,E1 31268.042,E2 31268.042} C_VEL
LIN {X 0,Y 714.126,Z 489.605,A -85,B 0,C 180,E1 31267.581,E2 31267.581} C_VEL
LIN {X 0,Y 718.324,Z 500.283,A -85,B 0,C 180,E1 31266.665,E2 31266.665} C_VEL
LIN {X 0,Y 717.894,Z 528.369,A -85,B 0,C 180,E1 31265.009,E2 31265.009} C_VEL
LIN {X 0,Y 719.863,Z 538.722,A -85,B 0,C 180,E1 31264.769,E2 31264.769} C_VEL
LIN {X 0,Y 718.587,Z 795.359,A -85,B 0,C 180,E1 31261.832,E2 31261.832} C_VEL
LIN {X 0,Y 718.005,Z 919.153,A -85,B 0,C 180,E1 31260.419,E2 31260.419} C_VEL
LIN {X 0,Y 717.628,Z 944.817,A -85,B 0,C 180,E1 31259.981,E2 31259.981} C_VEL
LIN {X 0,Y 717.289,Z 966.502,A -85,B 0,C 180,E1 31259.473,E2 31259.473} C_VEL
LIN {X 0,Y 716.865,Z 990.598,A -85,B 0,C 180,E1 31258.763,E2 31258.763} C_VEL
LIN {X 0,Y 716.34,Z 1012.512,A -85,B 0,C 180,E1 31257.968,E2 31257.968} C_VEL
LIN {X 0,Y 715.832,Z 1035.579,A -85,B 0,C 180,E1 31256.978,E2 31256.978} C_VEL
LIN {X 0,Y 715.249,Z 1056.773,A -85,B 0,C 180,E1 31255.903,E2 31255.903} C_VEL
LIN {X 0,Y 714.718,Z 1077.769,A -85,B 0,C 180,E1 31254.682,E2 31254.682} C_VEL
LIN {X 0,Y 714.179,Z 1097.136,A -85,B 0,C 180,E1 31253.379,E2 31253.379} C_VEL
LIN {X 0,Y 713.72,Z 1115.818,A -85,B 0,C 180,E1 31251.961,E2 31251.961} C_VEL
LIN {X 0,Y 713.295,Z 1132.47,A -85,B 0,C 180,E1 31250.514,E2 31250.514} C_VEL
LIN {X 0,Y 712.946,Z 1148.972,A -85,B 0,C 180,E1 31248.903,E2 31248.903} C_VEL
LIN {X 0,Y 712.62,Z 1163.227,A -85,B 0,C 180,E1 31247.305,E2 31247.305} C_VEL
LIN {X 0,Y 712.389,Z 1177.064,A -85,B 0,C 180,E1 31245.55,E2 31245.55} C_VEL
LIN {X 0,Y 712.207,Z 1188.8,A -85,B 0,C 180,E1 31243.807,E2 31243.807} C_VEL
LIN {X 0,Y 712.078,Z 1198.951,A -85,B 0,C 180,E1 31242.076,E2 31242.076} C_VEL
LIN {X 0,Y 711.986,Z 1208.184,A -85,B 0,C 180,E1 31240.192,E2 31240.192} C_VEL
LIN {X 0,Y 711.945,Z 1214.817,A -85,B 0,C 180,E1 31238.561,E2 31238.561} C_VEL
LIN {X 0,Y 711.924,Z 1221.245,A -85,B 0,C 180,E1 31236.613,E2 31236.613} C_VEL
LIN {X 0,Y 711.914,Z 1225.814,A -85,B 0,C 180,E1 31234.672,E2 31234.672} C_VEL
LIN {X 0,Y 711.882,Z 1228.685,A -85,B 0,C 180,E1 31232.898,E2 31232.898} C_VEL
LIN {X 0,Y 711.891,Z 1230.262,A -85,B 0,C 180,E1 31230.885,E2 31230.885} C_VEL
LIN {X 0,Y 711.883,Z 1230.306,A -85,B 0,C 180,E1 31229.276,E2 31229.276} C_VEL
LIN {X 0,Y 711.888,Z 1229.017,A -85,B 0,C 180,E1 31227.343,E2 31227.343} C_VEL
LIN {X 0,Y 711.917,Z 1225.972,A -85,B 0,C 180,E1 31225.408,E2 31225.408} C_VEL
LIN {X 0,Y 711.924,Z 1221.865,A -85,B 0,C 180,E1 31223.63,E2 31223.63} C_VEL
LIN {X 0,Y 711.954,Z 1215.424,A -85,B 0,C 180,E1 31221.602,E2 31221.602} C_VEL
LIN {X 0,Y 711.97,Z 1208.894,A -85,B 0,C 180,E1 31219.971,E2 31219.971} C_VEL
LIN {X 0,Y 712.075,Z 1199.869,A -85,B 0,C 180,E1 31218.088,E2 31218.088} C_VEL
LIN {X 0,Y 712.198,Z 1189.321,A -85,B 0,C 180,E1 31216.275,E2 31216.275} C_VEL
LIN {X 0,Y 712.375,Z 1177.646,A -85,B 0,C 180,E1 31214.533,E2 31214.533} C_VEL
LIN {X 0,Y 712.606,Z 1163.934,A -85,B 0,C 180,E1 31212.779,E2 31212.779} C_VEL
LIN {X 0,Y 712.925,Z 1149.748,A -85,B 0,C 180,E1 31211.182,E2 31211.182} C_VEL
LIN {X 0,Y 713.269,Z 1133.399,A -85,B 0,C 180,E1 31209.571,E2 31209.571} C_VEL
LIN {X 0,Y 713.69,Z 1116.787,A -85,B 0,C 180,E1 31208.12,E2 31208.12} C_VEL
LIN {X 0,Y 714.164,Z 1097.665,A -85,B 0,C 180,E1 31206.659,E2 31206.659} C_VEL
LIN {X 0,Y 714.698,Z 1078.433,A -85,B 0,C 180,E1 31205.361,E2 31205.361} C_VEL
LIN {X 0,Y 715.221,Z 1057.572,A -85,B 0,C 180,E1 31204.141,E2 31204.141} C_VEL
LIN {X 0,Y 715.786,Z 1036.997,A -85,B 0,C 180,E1 31203.09,E2 31203.09} C_VEL
LIN {X 0,Y 716.315,Z 1013.72,A -85,B 0,C 180,E1 31202.079,E2 31202.079} C_VEL
LIN {X 0,Y 716.786,Z 993.167,A -85,B 0,C 180,E1 31201.324,E2 31201.324} C_VEL
LIN {X 0,Y 717.276,Z 968.162,A -85,B 0,C 180,E1 31200.571,E2 31200.571} C_VEL
LIN {X 0,Y 717.596,Z 946.643,A -85,B 0,C 180,E1 31200.058,E2 31200.058} C_VEL
LIN {X 0,Y 717.993,Z 921.509,A -85,B 0,C 180,E1 31199.612,E2 31199.612} C_VEL
LIN {X 0,Y 718.273,Z 868.392,A -85,B 0,C 180,E1 31198.99,E2 31198.99} C_VEL
LIN {X 0,Y 719.349,Z 632.367,A -85,B 0,C 180,E1 31196.31,E2 31196.31} C_VEL
LIN {X 0,Y 719.67,Z 536.827,A -85,B 0,C 180,E1 31195.197,E2 31195.197} C_VEL
LIN {X 0,Y 717.835,Z 527.989,A -85,B 0,C 180,E1 31194.98,E2 31194.98} C_VEL
LIN {X 0,Y 718.277,Z 499.853,A -85,B 0,C 180,E1 31193.306,E2 31193.306} C_VEL
LIN {X 0,Y 712.276,Z 484.853,A -85,B 0,C 180,E1 31191.983,E2 31191.983} C_VEL
LIN {X 0,Y 712.233,Z 484.504,A -85,B 0,C 180,E1 31191.312,E2 31191.312} C_VEL
LIN {X 0,Y 712.27,Z 484.494,A -85,B 0,C 180,E1 31188.288,E2 31188.288} C_VEL
LIN {X 0,Y 712.219,Z 484.508,A -85,B 0,C 180,E1 31185.495,E2 31185.495} C_VEL
LIN {X 0,Y 712.273,Z 484.495,A -85,B 0,C 180,E1 31182.691,E2 31182.691} C_VEL
LIN {X 0,Y 712.235,Z 484.494,A -85,B 0,C 180,E1 31179.7,E2 31179.7} C_VEL
